gfCNCPoint5[16848] = {X 82.2240, Y 14.7584, Z -7.1667, A 0.000, B 0.000, C 0.000 }
gfCNCPoint5[16849] = {X 81.9226, Y 13.9083, Z -7.1667, A 0.000, B 0.000, C 0.000 }
gfCNCPoint5[16850] = {X 81.8152, Y 13.0128, Z -7.1667, A 0.000, B 0.000, C 0.000 }
gfCNCPoint5[16851] = {X 81.8151, Y 12.1868, Z -7.1667, A 0.000, B 0.000, C 0.000 }
gfCNCPoint5[16852] = {X 81.9174, Y 11.2789, Z -7.1667, A 0.000, B 0.000, C 0.000 }
gfCNCPoint5[16853] = {X 82.2191, Y 10.4166, Z -7.1667, A 0.000, B 0.000, C 0.000 }
gfCNCPoint5[16854] = {X 82.7052, Y 9.6430, Z -7.1667, A 0.000, B 0.000, C 0.000 }
gfCNCPoint5[16855] = {X 83.3512, Y 8.9969, Z -7.1667, A 0.000, B 0.000, C 0.000 }
gfCNCPoint5[16856] = {X 84.1248, Y 8.5109, Z -7.1667, A 0.000, B 0.000, C 0.000 }
gfCNCPoint5[16857] = {X 84.9872, Y 8.2091, Z -7.1667, A 0.000, B 0.000, C 0.000 }
gfCNCPoint5[16858] = {X 85.8951, Y 8.1068, Z -7.1667, A 0.000, B 0.000, C 0.000 }
gfCNCPoint5[16859] = {X 94.0497, Y 8.1068, Z -7.1667, A 0.000, B 0.000, C 0.000 }
gfCNCPoint5[16860] = {X 94.9576, Y 8.2091, Z -7.1667, A 0.000, B 0.000, C 0.000 }
gfCNCPoint5[16861] = {X 95.8199, Y 8.5109, Z -7.1667, A 0.000, B 0.000, C 0.000 }
gfCNCPoint5[16862] = {X 96.5935, Y 8.9969, Z -7.1667, A 0.000, B 0.000, C 0.000 }
gfCNCPoint5[16863] = {X 97.2395, Y 9.6430, Z -7.1667, A 0.000, B 0.000, C 0.000 }
gfCNCPoint5[16864] = {X 97.7256, Y 10.4166, Z -7.1667, A 0.000, B 0.000, C 0.000 }
gfCNCPoint5[16865] = {X 98.0274, Y 11.2789, Z -7.1667, A 0.000, B 0.000, C 0.000 }
gfCNCPoint5[16866] = {X 98.1297, Y 12.1868, Z -7.1667, A 0.000, B 0.000, C 0.000 }
gfCNCPoint5[16867] = {X 98.1297, Y 12.9782, Z -7.1667, A 0.000, B 0.000, C 0.000 }
gfCNCPoint5[16868] = {X 98.0632, Y 13.7116, Z -7.1667, A 0.000, B 0.000, C 0.000 }
gfCNCPoint5[16869] = {X 97.8659, Y 14.4211, Z -7.1667, A 0.000, B 0.000, C 0.000 }
gfCNCPoint5[16870] = {X 97.5443, Y 15.0836, Z -7.1667, A 0.000, B 0.000, C 0.000 }
gfCNCPoint5[16871] = {X 97.4977, Y 15.1591, Z -7.1667, A 0.000, B 0.000, C 0.000 }
gfCNCPoint5[16872] = {X 97.4495, Y 15.2336, Z -7.1667, A 0.000, B 0.000, C 0.000 }
gfCNCPoint5[16873] = {X 97.4864, Y 15.2810, Z -7.1667, A 0.000, B 0.000, C 0.000 }
gfCNCPoint5[16874] = {X 101.8776, Y 26.1666, Z -7.1667, A 0.000, B 0.000, C 0.000 }
gfCNCPoint5[16875] = {X 106.2844, Y 15.1969, Z -7.1667, A 0.000, B 0.000, C 0.000 }
gfCNCPoint5[16876] = {X 106.2408, Y 15.1282, Z -7.1667, A 0.000, B 0.000, C 0.000 }
gfCNCPoint5[16877] = {X 106.1986, Y 15.0586, Z -7.1667, A 0.000, B 0.000, C 0.000 }
gfCNCPoint5[16878] = {X 105.8896, Y 14.4146, Z -7.1667, A 0.000, B 0.000, C 0.000 }
gfCNCPoint5[16879] = {X 105.6975, Y 13.7266, Z -7.1667, A 0.000, B 0.000, C 0.000 }
gfCNCPoint5[16880] = {X 105.6285, Y 13.0157, Z -7.1667, A 0.000, B 0.000, C 0.000 }
gfCNCPoint5[16881] = {X 105.6283, Y 12.1868, Z -7.1667, A 0.000, B 0.000, C 0.000 }
gfCNCPoint5[16882] = {X 105.7306, Y 11.2789, Z -7.1667, A 0.000, B 0.000, C 0.000 }
gfCNCPoint5[16883] = {X 106.0323, Y 10.4166, Z -7.1667, A 0.000, B 0.000, C 0.000 }
gfCNCPoint5[16884] = {X 106.5184, Y 9.6430, Z -7.1667, A 0.000, B 0.000, C 0.000 }
gfCNCPoint5[16885] = {X 107.1644, Y 8.9969, Z -7.1667, A 0.000, B 0.000, C 0.000 }
gfCNCPoint5[16886] = {X 107.9380, Y 8.5109, Z -7.1667, A 0.000, B 0.000, C 0.000 }
gfCNCPoint5[16887] = {X 108.8004, Y 8.2091, Z -7.1667, A 0.000, B 0.000, C 0.000 }
gfCNCPoint5[16888] = {X 109.7083, Y 8.1068, Z -7.1667, A 0.000, B 0.000, C 0.000 }
gfCNCPoint5[16889] = {X 117.7916, Y 8.1068, Z -7.1667, A 0.000, B 0.000, C 0.000 }
gfCNCPoint5[16890] = {X 118.6995, Y 8.2091, Z -7.1667, A 0.000, B 0.000, C 0.000 }
gfCNCPoint5[16891] = {X 119.5618, Y 8.5109, Z -7.1667, A 0.000, B 0.000, C 0.000 }
gfCNCPoint5[16892] = {X 120.3354, Y 8.9969, Z -7.1667, A 0.000, B 0.000, C 0.000 }
gfCNCPoint5[16893] = {X 120.9814, Y 9.6430, Z -7.1667, A 0.000, B 0.000, C 0.000 }
gfCNCPoint5[16894] = {X 121.4675, Y 10.4166, Z -7.1667, A 0.000, B 0.000, C 0.000 }
gfCNCPoint5[16895] = {X 121.7693, Y 11.2789, Z -7.1667, A 0.000, B 0.000, C 0.000 }
gfCNCPoint5[16896] = {X 121.8716, Y 12.1868, Z -7.1667, A 0.000, B 0.000, C 0.000 }
gfCNCPoint5[16897] = {X 121.8716, Y 12.9782, Z -7.1667, A 0.000, B 0.000, C 0.000 }
gfCNCPoint5[16898] = {X 121.7699, Y 13.8830, Z -7.1667, A 0.000, B 0.000, C 0.000 }
gfCNCPoint5[16899] = {X 121.4702, Y 14.7427, Z -7.1667, A 0.000, B 0.000, C 0.000 }
gfCNCPoint5[16900] = {X 120.9872, Y 15.5146, Z -7.1667, A 0.000, B 0.000, C 0.000 }
gfCNCPoint5[16901] = {X 120.3451, Y 16.1601, Z -7.1667, A 0.000, B 0.000, C 0.000 }
gfCNCPoint5[16902] = {X 120.3450, Y 41.0278, Z -7.1667, A 0.000, B 0.000, C 0.000 }
gfCNCPoint5[16903] = {X 120.4677, Y 41.1291, Z -7.1667, A 0.000, B 0.000, C 0.000 }
gfCNCPoint5[16904] = {X 121.0553, Y 41.7605, Z -7.1667, A 0.000, B 0.000, C 0.000 }
gfCNCPoint5[16905] = {X 121.4971, Y 42.5013, Z -7.1667, A 0.000, B 0.000, C 0.000 }
gfCNCPoint5[16906] = {X 121.7732, Y 43.3184, Z -7.1667, A 0.000, B 0.000, C 0.000 }
gfCNCPoint5[16907] = {X 121.8714, Y 44.1754, Z -7.1667, A 0.000, B 0.000, C 0.000 }
gfCNCPoint5[16908] = {X 121.8716, Y 45.0000, Z -7.1667, A 0.000, B 0.000, C 0.000 }
gfCNCPoint5[16909] = {X 121.7693, Y 45.9079, Z -7.1667, A 0.000, B 0.000, C 0.000 }
gfCNCPoint5[16910] = {X 121.4675, Y 46.7702, Z -7.1667, A 0.000, B 0.000, C 0.000 }
gfCNCPoint5[16911] = {X 120.9814, Y 47.5438, Z -7.1667, A 0.000, B 0.000, C 0.000 }
gfCNCPoint5[16912] = {X 120.3354, Y 48.1899, Z -7.1667, A 0.000, B 0.000, C 0.000 }
gfCNCPoint5[16913] = {X 119.5618, Y 48.6760, Z -7.1667, A 0.000, B 0.000, C 0.000 }
gfCNCPoint5[16914] = {X 118.6995, Y 48.9777, Z -7.1667, A 0.000, B 0.000, C 0.000 }
gfCNCPoint5[16915] = {X 117.7916, Y 49.0800, Z -7.1667, A 0.000, B 0.000, C 0.000 }
gfCNCPoint5[16916] = {X 111.9185, Y 49.0800, Z -7.1667, A 0.000, B 0.000, C 0.000 }
gfCNCPoint5[16917] = {X 111.0151, Y 48.9787, Z -7.1667, A 0.000, B 0.000, C 0.000 }
gfCNCPoint5[16918] = {X 110.1565, Y 48.6799, Z -7.1667, A 0.000, B 0.000, C 0.000 }
gfCNCPoint5[16919] = {X 109.3855, Y 48.1985, Z -7.1667, A 0.000, B 0.000, C 0.000 }
gfCNCPoint5[16920] = {X 108.7401, Y 47.5582, Z -7.1667, A 0.000, B 0.000, C 0.000 }
gfCNCPoint5[16921] = {X 108.2526, Y 46.7909, Z -7.1667, A 0.000, B 0.000, C 0.000 }
gfCNCPoint5[16922] = {X 107.9470, Y 45.9348, Z -7.1667, A 0.000, B 0.000, C 0.000 }
gfCNCPoint5[16923] = {X 107.8386, Y 45.0322, Z -7.1667, A 0.000, B 0.000, C 0.000 }
gfCNCPoint5[16924] = {X 107.8385, Y 44.1771, Z -7.1667, A 0.000, B 0.000, C 0.000 }
gfCNCPoint5[16925] = {X 107.8717, Y 43.6680, Z -7.1667, A 0.000, B 0.000, C 0.000 }
gfCNCPoint5[16926] = {X 107.9710, Y 43.1676, Z -7.1667, A 0.000, B 0.000, C 0.000 }
gfCNCPoint5[16927] = {X 108.1299, Y 42.6955, Z -7.1667, A 0.000, B 0.000, C 0.000 }
gfCNCPoint5[16928] = {X 108.3475, Y 42.2474, Z -7.1667, A 0.000, B 0.000, C 0.000 }
gfCNCPoint5[16929] = {X 108.8090, Y 41.5687, Z -7.1667, A 0.000, B 0.000, C 0.000 }
gfCNCPoint5[16930] = {X 109.3649, Y 40.9650, Z -7.1667, A 0.000, B 0.000, C 0.000 }
gfCNCPoint5[16931] = {X 109.3648, Y 39.0029, Z -7.1667, A 0.000, B 0.000, C 0.000 }
gfCNCPoint5[16932] = {X 108.9865, Y 39.0029, Z -7.1667, A 0.000, B 0.000, C 0.000 }
gfCNCPoint5[16933] = {X 105.8902, Y 46.5692, Z -7.1667, A 0.000, B 0.000, C 0.000 }
gfCNCPoint5[16934] = {X 105.5407, Y 47.2300, Z -7.1667, A 0.000, B 0.000, C 0.000 }
gfCNCPoint5[16935] = {X 105.0765, Y 47.8159, Z -7.1667, A 0.000, B 0.000, C 0.000 }
gfCNCPoint5[16936] = {X 104.5133, Y 48.3073, Z -7.1667, A 0.000, B 0.000, C 0.000 }
gfCNCPoint5[16937] = {X 103.8698, Y 48.6877, Z -7.1667, A 0.000, B 0.000, C 0.000 }
gfCNCPoint5[16938] = {X 102.9784, Y 48.9895, Z -7.1667, A 0.000, B 0.000, C 0.000 }
gfCNCPoint5[16939] = {X 102.0417, Y 49.0792, Z -7.1667, A 0.000, B 0.000, C 0.000 }
gfCNCPoint5[16940] = {X 101.1093, Y 48.9518, Z -7.1667, A 0.000, B 0.000, C 0.000 }
gfCNCPoint5[16941] = {X 100.2309, Y 48.6142, Z -7.1667, A 0.000, B 0.000, C 0.000 }
gfCNCPoint5[16942] = {X 99.4532, Y 48.0843, Z -7.1667, A 0.000, B 0.000, C 0.000 }
gfCNCPoint5[16943] = {X 98.8176, Y 47.3903, Z -7.1667, A 0.000, B 0.000, C 0.000 }
gfCNCPoint5[16944] = {X 98.3579, Y 46.5692, Z -7.1667, A 0.000, B 0.000, C 0.000 }
gfCNCPoint5[16945] = {X 94.8929, Y 38.0952, Z -7.1667, A 0.000, B 0.000, C 0.000 }
gfCNCPoint5[16946] = {X 94.8920, Y 38.2309, Z -7.1667, A 0.000, B 0.000, C 0.000 }
gfCNCPoint5[16947] = {X 94.8920, Y 41.0165, Z -7.1667, A 0.000, B 0.000, C 0.000 }
gfCNCPoint5[16948] = {X 95.4369, Y 41.5527, Z -7.1667, A 0.000, B 0.000, C 0.000 }
gfCNCPoint5[16949] = {X 95.8744, Y 42.1796, Z -7.1667, A 0.000, B 0.000, C 0.000 }
gfCNCPoint5[16950] = {X 96.1092, Y 42.6624, Z -7.1667, A 0.000, B 0.000, C 0.000 }
gfCNCPoint5[16951] = {X 96.2799, Y 43.1714, Z -7.1667, A 0.000, B 0.000, C 0.000 }
gfCNCPoint5[16952] = {X 96.3820, Y 43.6855, Z -7.1667, A 0.000, B 0.000, C 0.000 }
gfCNCPoint5[16953] = {X 96.4185, Y 44.2083, Z -7.1667, A 0.000, B 0.000, C 0.000 }
gfCNCPoint5[16954] = {X 96.4184, Y 45.0392, Z -7.1667, A 0.000, B 0.000, C 0.000 }
gfCNCPoint5[16955] = {X 96.3086, Y 45.9406, Z -7.1667, A 0.000, B 0.000, C 0.000 }
gfCNCPoint5[16956] = {X 96.0023, Y 46.7954, Z -7.1667, A 0.000, B 0.000, C 0.000 }
gfCNCPoint5[16957] = {X 95.5144, Y 47.5613, Z -7.1667, A 0.000, B 0.000, C 0.000 }
gfCNCPoint5[16958] = {X 94.8692, Y 48.2003, Z -7.1667, A 0.000, B 0.000, C 0.000 }
gfCNCPoint5[16959] = {X 94.0987, Y 48.6808, Z -7.1667, A 0.000, B 0.000, C 0.000 }
gfCNCPoint5[16960] = {X 93.2410, Y 48.9789, Z -7.1667, A 0.000, B 0.000, C 0.000 }
gfCNCPoint5[16961] = {X 92.3385, Y 49.0800, Z -7.1667, A 0.000, B 0.000, C 0.000 }
gfCNCPoint5[16962] = {X 85.8951, Y 49.0800, Z -7.1667, A 0.000, B 0.000, C 0.000 }
gfCNCPoint5[16963] = {X 84.9918, Y 48.9788, Z -7.1667, A 0.000, B 0.000, C 0.000 }
gfCNCPoint5[16964] = {X 84.1334, Y 48.6801, Z -7.1667, A 0.000, B 0.000, C 0.000 }
gfCNCPoint5[16965] = {X 83.3624, Y 48.1987, Z -7.1667, A 0.000, B 0.000, C 0.000 }
gfCNCPoint5[16966] = {X 82.7171, Y 47.5586, Z -7.1667, A 0.000, B 0.000, C 0.000 }
gfCNCPoint5[16967] = {X 82.2295, Y 46.7916, Z -7.1667, A 0.000, B 0.000, C 0.000 }
gfCNCPoint5[16968] = {X 81.9238, Y 45.9356, Z -7.1667, A 0.000, B 0.000, C 0.000 }
gfCNCPoint5[16969] = {X 81.8152, Y 45.0332, Z -7.1667, A 0.000, B 0.000, C 0.000 }
gfCNCPoint5[16970] = {X 81.8151, Y 44.2084, Z -7.1667, A 0.000, B 0.000, C 0.000 }
gfCNCPoint5[16971] = {X 81.9200, Y 43.3034, Z -7.1667, A 0.000, B 0.000, C 0.000 }
gfCNCPoint5[16972] = {X 82.2207, Y 42.4433, Z -7.1667, A 0.000, B 0.000, C 0.000 }
gfCNCPoint5[16973] = {X 82.7024, Y 41.6699, Z -7.1667, A 0.000, B 0.000, C 0.000 }
gfCNCPoint5[16974] = {X 83.3419, Y 41.0209, Z -7.1667, A 0.000, B 0.000, C 0.000 }
gfCNCPoint5[16975] = {X 83.3418, Y 28.5910, Z -7.1667, A 0.000, B 0.000, C 0.000 }
gfCNCPoint5[16976] = {X 79.3418, Y 28.5910, Z -7.1667, A 0.000, B 0.000, C 0.000 }
gfCNCPoint5[16977] = {X 83.4218, Y 28.5910, Z -7.1667, A 0.000, B 0.000, C 0.000 }
gfCNCPoint5[16978] = {X 83.4217, Y 16.1216, Z -7.1667, A 0.000, B 0.000, C 0.000 }
gfCNCPoint5[16979] = {X 82.7800, Y 15.4873, Z -7.1667, A 0.000, B 0.000, C 0.000 }
gfCNCPoint5[16980] = {X 82.2969, Y 14.7253, Z -7.1667, A 0.000, B 0.000, C 0.000 }
gfCNCPoint5[16981] = {X 81.9968, Y 13.8745, Z -7.1667, A 0.000, B 0.000, C 0.000 }
gfCNCPoint5[16982] = {X 81.8951, Y 12.9780, Z -7.1667, A 0.000, B 0.000, C 0.000 }
gfCNCPoint5[16983] = {X 81.8951, Y 12.1868, Z -7.1667, A 0.000, B 0.000, C 0.000 }
gfCNCPoint5[16984] = {X 81.9954, Y 11.2967, Z -7.1667, A 0.000, B 0.000, C 0.000 }
gfCNCPoint5[16985] = {X 82.2912, Y 10.4513, Z -7.1667, A 0.000, B 0.000, C 0.000 }
gfCNCPoint5[16986] = {X 82.7677, Y 9.6929, Z -7.1667, A 0.000, B 0.000, C 0.000 }
gfCNCPoint5[16987] = {X 83.4011, Y 9.0595, Z -7.1667, A 0.000, B 0.000, C 0.000 }
gfCNCPoint5[16988] = {X 84.1595, Y 8.5829, Z -7.1667, A 0.000, B 0.000, C 0.000 }
gfCNCPoint5[16989] = {X 85.0050, Y 8.2871, Z -7.1667, A 0.000, B 0.000, C 0.000 }
gfCNCPoint5[16990] = {X 85.8951, Y 8.1868, Z -7.1667, A 0.000, B 0.000, C 0.000 }
gfCNCPoint5[16991] = {X 94.0497, Y 8.1868, Z -7.1667, A 0.000, B 0.000, C 0.000 }
gfCNCPoint5[16992] = {X 94.9398, Y 8.2871, Z -7.1667, A 0.000, B 0.000, C 0.000 }
gfCNCPoint5[16993] = {X 95.7852, Y 8.5829, Z -7.1667, A 0.000, B 0.000, C 0.000 }
gfCNCPoint5[16994] = {X 96.5436, Y 9.0595, Z -7.1667, A 0.000, B 0.000, C 0.000 }
gfCNCPoint5[16995] = {X 97.1770, Y 9.6929, Z -7.1667, A 0.000, B 0.000, C 0.000 }
gfCNCPoint5[16996] = {X 97.6535, Y 10.4513, Z -7.1667, A 0.000, B 0.000, C 0.000 }
gfCNCPoint5[16997] = {X 97.9494, Y 11.2967, Z -7.1667, A 0.000, B 0.000, C 0.000 }
gfCNCPoint5[16998] = {X 98.0497, Y 12.1868, Z -7.1667, A 0.000, B 0.000, C 0.000 }
gfCNCPoint5[16999] = {X 98.0495, Y 13.0192, Z -7.1667, A 0.000, B 0.000, C 0.000 }
gfCNCPoint5[17000] = {X 97.9795, Y 13.7241, Z -7.1667, A 0.000, B 0.000, C 0.000 }
gfCNCPoint5[17001] = {X 97.7862, Y 14.4056, Z -7.1667, A 0.000, B 0.000, C 0.000 }
gfCNCPoint5[17002] = {X 97.4758, Y 15.0424, Z -7.1667, A 0.000, B 0.000, C 0.000 }
gfCNCPoint5[17003] = {X 97.4132, Y 15.1429, Z -7.1667, A 0.000, B 0.000, C 0.000 }
gfCNCPoint5[17004] = {X 97.3476, Y 15.2415, Z -7.1667, A 0.000, B 0.000, C 0.000 }
gfCNCPoint5[17005] = {X 97.4122, Y 15.3109, Z -7.1667, A 0.000, B 0.000, C 0.000 }
gfCNCPoint5[17006] = {X 101.8768, Y 26.3785, Z -7.1667, A 0.000, B 0.000, C 0.000 }
gfCNCPoint5[17007] = {X 101.9496, Y 26.2020, Z -7.1667, A 0.000, B 0.000, C 0.000 }
gfCNCPoint5[17008] = {X 105.4120, Y 17.5683, Z -7.1667, A 0.000, B 0.000, C 0.000 }
gfCNCPoint5[17009] = {X 106.3409, Y 15.2554, Z -7.1667, A 0.000, B 0.000, C 0.000 }
gfCNCPoint5[17010] = {X 106.3813, Y 15.1986, Z -7.1667, A 0.000, B 0.000, C 0.000 }
gfCNCPoint5[17011] = {X 106.3231, Y 15.1090, Z -7.1667, A 0.000, B 0.000, C 0.000 }
gfCNCPoint5[17012] = {X 106.2675, Y 15.0178, Z -7.1667, A 0.000, B 0.000, C 0.000 }
gfCNCPoint5[17013] = {X 105.9601, Y 14.3749, Z -7.1667, A 0.000, B 0.000, C 0.000 }
gfCNCPoint5[17014] = {X 105.7717, Y 13.6877, Z -7.1667, A 0.000, B 0.000, C 0.000 }
gfCNCPoint5[17015] = {X 105.7083, Y 12.9780, Z -7.1667, A 0.000, B 0.000, C 0.000 }
gfCNCPoint5[17016] = {X 105.7083, Y 12.1868, Z -7.1667, A 0.000, B 0.000, C 0.000 }
gfCNCPoint5[17017] = {X 105.8086, Y 11.2967, Z -7.1667, A 0.000, B 0.000, C 0.000 }
gfCNCPoint5[17018] = {X 106.1044, Y 10.4513, Z -7.1667, A 0.000, B 0.000, C 0.000 }
gfCNCPoint5[17019] = {X 106.5810, Y 9.6929, Z -7.1667, A 0.000, B 0.000, C 0.000 }
gfCNCPoint5[17020] = {X 107.2143, Y 9.0595, Z -7.1667, A 0.000, B 0.000, C 0.000 }
gfCNCPoint5[17021] = {X 107.9727, Y 8.5829, Z -7.1667, A 0.000, B 0.000, C 0.000 }
gfCNCPoint5[17022] = {X 108.8182, Y 8.2871, Z -7.1667, A 0.000, B 0.000, C 0.000 }
gfCNCPoint5[17023] = {X 109.7083, Y 8.1868, Z -7.1667, A 0.000, B 0.000, C 0.000 }
gfCNCPoint5[17024] = {X 117.7916, Y 8.1868, Z -7.1667, A 0.000, B 0.000, C 0.000 }
gfCNCPoint5[17025] = {X 118.6817, Y 8.2871, Z -7.1667, A 0.000, B 0.000, C 0.000 }
gfCNCPoint5[17026] = {X 119.5271, Y 8.5829, Z -7.1667, A 0.000, B 0.000, C 0.000 }
gfCNCPoint5[17027] = {X 120.2855, Y 9.0595, Z -7.1667, A 0.000, B 0.000, C 0.000 }
gfCNCPoint5[17028] = {X 120.9189, Y 9.6929, Z -7.1667, A 0.000, B 0.000, C 0.000 }
gfCNCPoint5[17029] = {X 121.3955, Y 10.4513, Z -7.1667, A 0.000, B 0.000, C 0.000 }
gfCNCPoint5[17030] = {X 121.6913, Y 11.2967, Z -7.1667, A 0.000, B 0.000, C 0.000 }
gfCNCPoint5[17031] = {X 121.7916, Y 12.1868, Z -7.1667, A 0.000, B 0.000, C 0.000 }
gfCNCPoint5[17032] = {X 121.7914, Y 13.0192, Z -7.1667, A 0.000, B 0.000, C 0.000 }
gfCNCPoint5[17033] = {X 121.6828, Y 13.9045, Z -7.1667, A 0.000, B 0.000, C 0.000 }
gfCNCPoint5[17034] = {X 121.3807, Y 14.7438, Z -7.1667, A 0.000, B 0.000, C 0.000 }
gfCNCPoint5[17035] = {X 120.9002, Y 15.4952, Z -7.1667, A 0.000, B 0.000, C 0.000 }
gfCNCPoint5[17036] = {X 120.2651, Y 16.1215, Z -7.1667, A 0.000, B 0.000, C 0.000 }
gfCNCPoint5[17037] = {X 120.2650, Y 41.0655, Z -7.1667, A 0.000, B 0.000, C 0.000 }
gfCNCPoint5[17038] = {X 120.4160, Y 41.1901, Z -7.1667, A 0.000, B 0.000, C 0.000 }
gfCNCPoint5[17039] = {X 120.9967, Y 41.8157, Z -7.1667, A 0.000, B 0.000, C 0.000 }
gfCNCPoint5[17040] = {X 121.4315, Y 42.5502, Z -7.1667, A 0.000, B 0.000, C 0.000 }
gfCNCPoint5[17041] = {X 121.7005, Y 43.3602, Z -7.1667, A 0.000, B 0.000, C 0.000 }
gfCNCPoint5[17042] = {X 121.7916, Y 44.2089, Z -7.1667, A 0.000, B 0.000, C 0.000 }
gfCNCPoint5[17043] = {X 121.7916, Y 45.0000, Z -7.1667, A 0.000, B 0.000, C 0.000 }
gfCNCPoint5[17044] = {X 121.6913, Y 45.8901, Z -7.1667, A 0.000, B 0.000, C 0.000 }
gfCNCPoint5[17045] = {X 121.3955, Y 46.7355, Z -7.1667, A 0.000, B 0.000, C 0.000 }
gfCNCPoint5[17046] = {X 120.9189, Y 47.4940, Z -7.1667, A 0.000, B 0.000, C 0.000 }
gfCNCPoint5[17047] = {X 120.2855, Y 48.1273, Z -7.1667, A 0.000, B 0.000, C 0.000 }
gfCNCPoint5[17048] = {X 119.5271, Y 48.6039, Z -7.1667, A 0.000, B 0.000, C 0.000 }
gfCNCPoint5[17049] = {X 118.6817, Y 48.8997, Z -7.1667, A 0.000, B 0.000, C 0.000 }
gfCNCPoint5[17050] = {X 117.7916, Y 49.0000, Z -7.1667, A 0.000, B 0.000, C 0.000 }
gfCNCPoint5[17051] = {X 111.9185, Y 49.0000, Z -7.1667, A 0.000, B 0.000, C 0.000 }
gfCNCPoint5[17052] = {X 111.0284, Y 48.8997, Z -7.1667, A 0.000, B 0.000, C 0.000 }
gfCNCPoint5[17053] = {X 110.1829, Y 48.6039, Z -7.1667, A 0.000, B 0.000, C 0.000 }
gfCNCPoint5[17054] = {X 109.4245, Y 48.1273, Z -7.1667, A 0.000, B 0.000, C 0.000 }
gfCNCPoint5[17055] = {X 108.7911, Y 47.4939, Z -7.1667, A 0.000, B 0.000, C 0.000 }
gfCNCPoint5[17056] = {X 108.3146, Y 46.7355, Z -7.1667, A 0.000, B 0.000, C 0.000 }
gfCNCPoint5[17057] = {X 108.0188, Y 45.8901, Z -7.1667, A 0.000, B 0.000, C 0.000 }
gfCNCPoint5[17058] = {X 107.9185, Y 45.0000, Z -7.1667, A 0.000, B 0.000, C 0.000 }
gfCNCPoint5[17059] = {X 107.9185, Y 44.1771, Z -7.1667, A 0.000, B 0.000, C 0.000 }
gfCNCPoint5[17060] = {X 107.9511, Y 43.6784, Z -7.1667, A 0.000, B 0.000, C 0.000 }
gfCNCPoint5[17061] = {X 108.0483, Y 43.1883, Z -7.1667, A 0.000, B 0.000, C 0.000 }
gfCNCPoint5[17062] = {X 108.2039, Y 42.7258, Z -7.1667, A 0.000, B 0.000, C 0.000 }
gfCNCPoint5[17063] = {X 108.4171, Y 42.2868, Z -7.1667, A 0.000, B 0.000, C 0.000 }
gfCNCPoint5[17064] = {X 108.4423, Y 42.2431, Z -7.1667, A 0.000, B 0.000, C 0.000 }
gfCNCPoint5[17065] = {X 108.4680, Y 42.1997, Z -7.1667, A 0.000, B 0.000, C 0.000 }
gfCNCPoint5[17066] = {X 108.9141, Y 41.5653, Z -7.1667, A 0.000, B 0.000, C 0.000 }
gfCNCPoint5[17067] = {X 109.4449, Y 40.9999, Z -7.1667, A 0.000, B 0.000, C 0.000 }
gfCNCPoint5[17068] = {X 109.4448, Y 38.9229, Z -7.1667, A 0.000, B 0.000, C 0.000 }
gfCNCPoint5[17069] = {X 108.9328, Y 38.9229, Z -7.1667, A 0.000, B 0.000, C 0.000 }
gfCNCPoint5[17070] = {X 105.8164, Y 46.5384, Z -7.1667, A 0.000, B 0.000, C 0.000 }
gfCNCPoint5[17071] = {X 105.3339, Y 47.3869, Z -7.1667, A 0.000, B 0.000, C 0.000 }
gfCNCPoint5[17072] = {X 104.6602, Y 48.0932, Z -7.1667, A 0.000, B 0.000, C 0.000 }
gfCNCPoint5[17073] = {X 103.8355, Y 48.6154, Z -7.1667, A 0.000, B 0.000, C 0.000 }
gfCNCPoint5[17074] = {X 102.9580, Y 48.9121, Z -7.1667, A 0.000, B 0.000, C 0.000 }
gfCNCPoint5[17075] = {X 102.0357, Y 48.9990, Z -7.1667, A 0.000, B 0.000, C 0.000 }
gfCNCPoint5[17076] = {X 101.1182, Y 48.8715, Z -7.1667, A 0.000, B 0.000, C 0.000 }
gfCNCPoint5[17077] = {X 100.2546, Y 48.5362, Z -7.1667, A 0.000, B 0.000, C 0.000 }
gfCNCPoint5[17078] = {X 99.4912, Y 48.0114, Z -7.1667, A 0.000, B 0.000, C 0.000 }
gfCNCPoint5[17079] = {X 98.8691, Y 47.3250, Z -7.1667, A 0.000, B 0.000, C 0.000 }
gfCNCPoint5[17080] = {X 98.4216, Y 46.5139, Z -7.1667, A 0.000, B 0.000, C 0.000 }
gfCNCPoint5[17081] = {X 94.8156, Y 37.6948, Z -7.1667, A 0.000, B 0.000, C 0.000 }
gfCNCPoint5[17082] = {X 94.8120, Y 38.2306, Z -7.1667, A 0.000, B 0.000, C 0.000 }
gfCNCPoint5[17083] = {X 94.8120, Y 41.0546, Z -7.1667, A 0.000, B 0.000, C 0.000 }
gfCNCPoint5[17084] = {X 95.3635, Y 41.5899, Z -7.1667, A 0.000, B 0.000, C 0.000 }
gfCNCPoint5[17085] = {X 95.8049, Y 42.2191, Z -7.1667, A 0.000, B 0.000, C 0.000 }
gfCNCPoint5[17086] = {X 96.0352, Y 42.6926, Z -7.1667, A 0.000, B 0.000, C 0.000 }
gfCNCPoint5[17087] = {X 96.2026, Y 43.1919, Z -7.1667, A 0.000, B 0.000, C 0.000 }
gfCNCPoint5[17088] = {X 96.3027, Y 43.6961, Z -7.1667, A 0.000, B 0.000, C 0.000 }
gfCNCPoint5[17089] = {X 96.3385, Y 44.2089, Z -7.1667, A 0.000, B 0.000, C 0.000 }
gfCNCPoint5[17090] = {X 96.3384, Y 45.0384, Z -7.1667, A 0.000, B 0.000, C 0.000 }
gfCNCPoint5[17091] = {X 96.2308, Y 45.9222, Z -7.1667, A 0.000, B 0.000, C 0.000 }
gfCNCPoint5[17092] = {X 95.9304, Y 46.7602, Z -7.1667, A 0.000, B 0.000, C 0.000 }
gfCNCPoint5[17093] = {X 95.4521, Y 47.5111, Z -7.1667, A 0.000, B 0.000, C 0.000 }
gfCNCPoint5[17094] = {X 94.8196, Y 48.1376, Z -7.1667, A 0.000, B 0.000, C 0.000 }
gfCNCPoint5[17095] = {X 94.0642, Y 48.6086, Z -7.1667, A 0.000, B 0.000, C 0.000 }
gfCNCPoint5[17096] = {X 93.2233, Y 48.9009, Z -7.1667, A 0.000, B 0.000, C 0.000 }
gfCNCPoint5[17097] = {X 92.3385, Y 49.0000, Z -7.1667, A 0.000, B 0.000, C 0.000 }
gfCNCPoint5[17098] = {X 85.8951, Y 49.0000, Z -7.1667, A 0.000, B 0.000, C 0.000 }
gfCNCPoint5[17099] = {X 85.0050, Y 48.8997, Z -7.1667, A 0.000, B 0.000, C 0.000 }
gfCNCPoint5[17100] = {X 84.1595, Y 48.6039, Z -7.1667, A 0.000, B 0.000, C 0.000 }
gfCNCPoint5[17101] = {X 83.4011, Y 48.1273, Z -7.1667, A 0.000, B 0.000, C 0.000 }
gfCNCPoint5[17102] = {X 82.7677, Y 47.4939, Z -7.1667, A 0.000, B 0.000, C 0.000 }
gfCNCPoint5[17103] = {X 82.2912, Y 46.7355, Z -7.1667, A 0.000, B 0.000, C 0.000 }
gfCNCPoint5[17104] = {X 81.9954, Y 45.8901, Z -7.1667, A 0.000, B 0.000, C 0.000 }
gfCNCPoint5[17105] = {X 81.8951, Y 45.0000, Z -7.1667, A 0.000, B 0.000, C 0.000 }
gfCNCPoint5[17106] = {X 81.8951, Y 44.2088, Z -7.1667, A 0.000, B 0.000, C 0.000 }
gfCNCPoint5[17107] = {X 82.0001, Y 43.3120, Z -7.1667, A 0.000, B 0.000, C 0.000 }
gfCNCPoint5[17108] = {X 82.3011, Y 42.4607, Z -7.1667, A 0.000, B 0.000, C 0.000 }
gfCNCPoint5[17109] = {X 82.7829, Y 41.6972, Z -7.1667, A 0.000, B 0.000, C 0.000 }
gfCNCPoint5[17110] = {X 83.4219, Y 41.0592, Z -7.1667, A 0.000, B 0.000, C 0.000 }
gfCNCPoint5[17111] = {X 83.4218, Y 28.5910, Z -7.1667, A 0.000, B 0.000, C 0.000 }
gfCNCPoint5[17112] = {X 79.3418, Y 28.5910, Z -7.1667, A 0.000, B 0.000, C 0.000 }
gfCNCPoint5[17113] = {X 79.3418, Y 28.5910, Z -4.1667, A 0.000, B 0.000, C 0.000 }
gfCNCPoint5[17114] = {X 79.3418, Y 28.5910, Z 11.0000, A 0.000, B 0.000, C 0.000 }
gfCNCPoint5[17115] = {X 136.1636, Y 30.3969, Z 11.0000, A 0.000, B 0.000, C 0.000 }
gfCNCPoint5[17116] = {X 136.1636, Y 30.3969, Z -4.1667, A 0.000, B 0.000, C 0.000 }
gfCNCPoint5[17117] = {X 136.1636, Y 30.3969, Z -7.1667, A 0.000, B 0.000, C 0.000 }
gfCNCPoint5[17118] = {X 140.2436, Y 30.3969, Z -7.1667, A 0.000, B 0.000, C 0.000 }
gfCNCPoint5[17119] = {X 140.2436, Y 19.8782, Z -7.1667, A 0.000, B 0.000, C 0.000 }
gfCNCPoint5[17120] = {X 137.4233, Y 19.8779, Z -7.1667, A 0.000, B 0.000, C 0.000 }
gfCNCPoint5[17121] = {X 136.8909, Y 20.5223, Z -7.1667, A 0.000, B 0.000, C 0.000 }
gfCNCPoint5[17122] = {X 136.2444, Y 21.0521, Z -7.1667, A 0.000, B 0.000, C 0.000 }
gfCNCPoint5[17123] = {X 135.5079, Y 21.4475, Z -7.1667, A 0.000, B 0.000, C 0.000 }
gfCNCPoint5[17124] = {X 134.7091, Y 21.6937, Z -7.1667, A 0.000, B 0.000, C 0.000 }
gfCNCPoint5[17125] = {X 133.8778, Y 21.7814, Z -7.1667, A 0.000, B 0.000, C 0.000 }
gfCNCPoint5[17126] = {X 133.2006, Y 21.7815, Z -7.1667, A 0.000, B 0.000, C 0.000 }
gfCNCPoint5[17127] = {X 132.2394, Y 21.6732, Z -7.1667, A 0.000, B 0.000, C 0.000 }
gfCNCPoint5[17128] = {X 131.3263, Y 21.3537, Z -7.1667, A 0.000, B 0.000, C 0.000 }
gfCNCPoint5[17129] = {X 130.5072, Y 20.8390, Z -7.1667, A 0.000, B 0.000, C 0.000 }
gfCNCPoint5[17130] = {X 129.8231, Y 20.1550, Z -7.1667, A 0.000, B 0.000, C 0.000 }
gfCNCPoint5[17131] = {X 129.3085, Y 19.3359, Z -7.1667, A 0.000, B 0.000, C 0.000 }
gfCNCPoint5[17132] = {X 128.9890, Y 18.4228, Z -7.1667, A 0.000, B 0.000, C 0.000 }
gfCNCPoint5[17133] = {X 128.8806, Y 17.4615, Z -7.1667, A 0.000, B 0.000, C 0.000 }
gfCNCPoint5[17134] = {X 128.8806, Y 10.4835, Z -7.1667, A 0.000, B 0.000, C 0.000 }
gfCNCPoint5[17135] = {X 128.9874, Y 9.5289, Z -7.1667, A 0.000, B 0.000, C 0.000 }
gfCNCPoint5[17136] = {X 129.3026, Y 8.6214, Z -7.1667, A 0.000, B 0.000, C 0.000 }
gfCNCPoint5[17137] = {X 129.8104, Y 7.8061, Z -7.1667, A 0.000, B 0.000, C 0.000 }
gfCNCPoint5[17138] = {X 130.4859, Y 7.1231, Z -7.1667, A 0.000, B 0.000, C 0.000 }
gfCNCPoint5[17139] = {X 131.2956, Y 6.6063, Z -7.1667, A 0.000, B 0.000, C 0.000 }
gfCNCPoint5[17140] = {X 132.1995, Y 6.2811, Z -7.1667, A 0.000, B 0.000, C 0.000 }
gfCNCPoint5[17141] = {X 133.1529, Y 6.1638, Z -7.1667, A 0.000, B 0.000, C 0.000 }
gfCNCPoint5[17142] = {X 133.8866, Y 6.1637, Z -7.1667, A 0.000, B 0.000, C 0.000 }
gfCNCPoint5[17143] = {X 134.7108, Y 6.2517, Z -7.1667, A 0.000, B 0.000, C 0.000 }
gfCNCPoint5[17144] = {X 135.5031, Y 6.4955, Z -7.1667, A 0.000, B 0.000, C 0.000 }
gfCNCPoint5[17145] = {X 136.2342, Y 6.8861, Z -7.1667, A 0.000, B 0.000, C 0.000 }
gfCNCPoint5[17146] = {X 136.8772, Y 7.4091, Z -7.1667, A 0.000, B 0.000, C 0.000 }
gfCNCPoint5[17147] = {X 137.4085, Y 8.0454, Z -7.1667, A 0.000, B 0.000, C 0.000 }
gfCNCPoint5[17148] = {X 155.1133, Y 8.0467, Z -7.1667, A 0.000, B 0.000, C 0.000 }
gfCNCPoint5[17149] = {X 155.6453, Y 7.4093, Z -7.1667, A 0.000, B 0.000, C 0.000 }
gfCNCPoint5[17150] = {X 156.2894, Y 6.8855, Z -7.1667, A 0.000, B 0.000, C 0.000 }
gfCNCPoint5[17151] = {X 157.0219, Y 6.4946, Z -7.1667, A 0.000, B 0.000, C 0.000 }
gfCNCPoint5[17152] = {X 157.8156, Y 6.2510, Z -7.1667, A 0.000, B 0.000, C 0.000 }
gfCNCPoint5[17153] = {X 158.6412, Y 6.1637, Z -7.1667, A 0.000, B 0.000, C 0.000 }
gfCNCPoint5[17154] = {X 159.3781, Y 6.1639, Z -7.1667, A 0.000, B 0.000, C 0.000 }
gfCNCPoint5[17155] = {X 160.3301, Y 6.2828, Z -7.1667, A 0.000, B 0.000, C 0.000 }
gfCNCPoint5[17156] = {X 161.2324, Y 6.6088, Z -7.1667, A 0.000, B 0.000, C 0.000 }
gfCNCPoint5[17157] = {X 162.0405, Y 7.1260, Z -7.1667, A 0.000, B 0.000, C 0.000 }
gfCNCPoint5[17158] = {X 162.7145, Y 7.8088, Z -7.1667, A 0.000, B 0.000, C 0.000 }
gfCNCPoint5[17159] = {X 163.2212, Y 8.6236, Z -7.1667, A 0.000, B 0.000, C 0.000 }
gfCNCPoint5[17160] = {X 163.5355, Y 9.5300, Z -7.1667, A 0.000, B 0.000, C 0.000 }
gfCNCPoint5[17161] = {X 163.6421, Y 10.4835, Z -7.1667, A 0.000, B 0.000, C 0.000 }
gfCNCPoint5[17162] = {X 163.6421, Y 17.4615, Z -7.1667, A 0.000, B 0.000, C 0.000 }
gfCNCPoint5[17163] = {X 163.5355, Y 18.4152, Z -7.1667, A 0.000, B 0.000, C 0.000 }
gfCNCPoint5[17164] = {X 163.2211, Y 19.3218, Z -7.1667, A 0.000, B 0.000, C 0.000 }
gfCNCPoint5[17165] = {X 162.7142, Y 20.1366, Z -7.1667, A 0.000, B 0.000, C 0.000 }
gfCNCPoint5[17166] = {X 162.0400, Y 20.8194, Z -7.1667, A 0.000, B 0.000, C 0.000 }
gfCNCPoint5[17167] = {X 161.2318, Y 21.3365, Z -7.1667, A 0.000, B 0.000, C 0.000 }
gfCNCPoint5[17168] = {X 160.3292, Y 21.6625, Z -7.1667, A 0.000, B 0.000, C 0.000 }
gfCNCPoint5[17169] = {X 159.3770, Y 21.7812, Z -7.1667, A 0.000, B 0.000, C 0.000 }
gfCNCPoint5[17170] = {X 158.6794, Y 21.7815, Z -7.1667, A 0.000, B 0.000, C 0.000 }
gfCNCPoint5[17171] = {X 157.8410, Y 21.6970, Z -7.1667, A 0.000, B 0.000, C 0.000 }
gfCNCPoint5[17172] = {X 157.0346, Y 21.4525, Z -7.1667, A 0.000, B 0.000, C 0.000 }
gfCNCPoint5[17173] = {X 156.2904, Y 21.0570, Z -7.1667, A 0.000, B 0.000, C 0.000 }
gfCNCPoint5[17174] = {X 155.6365, Y 20.5255, Z -7.1667, A 0.000, B 0.000, C 0.000 }
gfCNCPoint5[17175] = {X 155.0973, Y 19.8779, Z -7.1667, A 0.000, B 0.000, C 0.000 }
gfCNCPoint5[17176] = {X 152.2772, Y 19.8789, Z -7.1667, A 0.000, B 0.000, C 0.000 }
gfCNCPoint5[17177] = {X 152.2761, Y 40.8742, Z -7.1667, A 0.000, B 0.000, C 0.000 }
gfCNCPoint5[17178] = {X 152.7408, Y 41.3745, Z -7.1667, A 0.000, B 0.000, C 0.000 }
gfCNCPoint5[17179] = {X 152.8367, Y 41.4887, Z -7.1667, A 0.000, B 0.000, C 0.000 }
gfCNCPoint5[17180] = {X 153.3624, Y 42.3140, Z -7.1667, A 0.000, B 0.000, C 0.000 }
gfCNCPoint5[17181] = {X 153.6900, Y 43.2360, Z -7.1667, A 0.000, B 0.000, C 0.000 }
gfCNCPoint5[17182] = {X 153.8031, Y 44.2079, Z -7.1667, A 0.000, B 0.000, C 0.000 }
gfCNCPoint5[17183] = {X 153.8029, Y 45.0415, Z -7.1667, A 0.000, B 0.000, C 0.000 }
gfCNCPoint5[17184] = {X 153.6867, Y 45.9960, Z -7.1667, A 0.000, B 0.000, C 0.000 }
gfCNCPoint5[17185] = {X 153.3623, Y 46.9011, Z -7.1667, A 0.000, B 0.000, C 0.000 }
gfCNCPoint5[17186] = {X 152.8458, Y 47.7120, Z -7.1667, A 0.000, B 0.000, C 0.000 }
gfCNCPoint5[17187] = {X 152.1626, Y 48.3886, Z -7.1667, A 0.000, B 0.000, C 0.000 }
gfCNCPoint5[17188] = {X 151.3468, Y 48.8973, Z -7.1667, A 0.000, B 0.000, C 0.000 }
gfCNCPoint5[17189] = {X 150.4386, Y 49.2130, Z -7.1667, A 0.000, B 0.000, C 0.000 }
gfCNCPoint5[17190] = {X 149.4831, Y 49.3200, Z -7.1667, A 0.000, B 0.000, C 0.000 }
gfCNCPoint5[17191] = {X 143.0396, Y 49.3200, Z -7.1667, A 0.000, B 0.000, C 0.000 }
gfCNCPoint5[17192] = {X 142.0831, Y 49.2128, Z -7.1667, A 0.000, B 0.000, C 0.000 }
gfCNCPoint5[17193] = {X 141.1741, Y 48.8964, Z -7.1667, A 0.000, B 0.000, C 0.000 }
gfCNCPoint5[17194] = {X 140.3576, Y 48.3866, Z -7.1667, A 0.000, B 0.000, C 0.000 }
gfCNCPoint5[17195] = {X 139.6743, Y 47.7087, Z -7.1667, A 0.000, B 0.000, C 0.000 }
gfCNCPoint5[17196] = {X 139.1581, Y 46.8964, Z -7.1667, A 0.000, B 0.000, C 0.000 }
gfCNCPoint5[17197] = {X 138.8346, Y 45.9899, Z -7.1667, A 0.000, B 0.000, C 0.000 }
gfCNCPoint5[17198] = {X 138.7198, Y 45.0342, Z -7.1667, A 0.000, B 0.000, C 0.000 }
gfCNCPoint5[17199] = {X 138.7200, Y 44.1494, Z -7.1667, A 0.000, B 0.000, C 0.000 }
gfCNCPoint5[17200] = {X 138.8305, Y 43.2364, Z -7.1667, A 0.000, B 0.000, C 0.000 }
gfCNCPoint5[17201] = {X 139.1317, Y 42.3675, Z -7.1667, A 0.000, B 0.000, C 0.000 }
gfCNCPoint5[17202] = {X 139.6099, Y 41.5821, Z -7.1667, A 0.000, B 0.000, C 0.000 }
gfCNCPoint5[17203] = {X 140.2436, Y 40.9157, Z -7.1667, A 0.000, B 0.000, C 0.000 }
gfCNCPoint5[17204] = {X 140.2436, Y 30.3969, Z -7.1667, A 0.000, B 0.000, C 0.000 }
gfCNCPoint5[17205] = {X 136.2436, Y 30.3969, Z -7.1667, A 0.000, B 0.000, C 0.000 }
gfCNCPoint5[17206] = {X 140.3236, Y 30.3969, Z -7.1667, A 0.000, B 0.000, C 0.000 }
gfCNCPoint5[17207] = {X 140.3236, Y 19.7982, Z -7.1667, A 0.000, B 0.000, C 0.000 }
gfCNCPoint5[17208] = {X 137.3793, Y 19.7979, Z -7.1667, A 0.000, B 0.000, C 0.000 }
gfCNCPoint5[17209] = {X 137.3564, Y 19.8340, Z -7.1667, A 0.000, B 0.000, C 0.000 }
gfCNCPoint5[17210] = {X 136.8339, Y 20.4662, Z -7.1667, A 0.000, B 0.000, C 0.000 }
gfCNCPoint5[17211] = {X 136.1994, Y 20.9860, Z -7.1667, A 0.000, B 0.000, C 0.000 }
gfCNCPoint5[17212] = {X 135.4767, Y 21.3739, Z -7.1667, A 0.000, B 0.000, C 0.000 }
gfCNCPoint5[17213] = {X 134.6928, Y 21.6154, Z -7.1667, A 0.000, B 0.000, C 0.000 }
gfCNCPoint5[17214] = {X 133.8772, Y 21.7014, Z -7.1667, A 0.000, B 0.000, C 0.000 }
gfCNCPoint5[17215] = {X 133.2006, Y 21.7015, Z -7.1667, A 0.000, B 0.000, C 0.000 }
gfCNCPoint5[17216] = {X 132.2572, Y 21.5952, Z -7.1667, A 0.000, B 0.000, C 0.000 }
gfCNCPoint5[17217] = {X 131.3610, Y 21.2816, Z -7.1667, A 0.000, B 0.000, C 0.000 }
gfCNCPoint5[17218] = {X 130.5570, Y 20.7765, Z -7.1667, A 0.000, B 0.000, C 0.000 }
gfCNCPoint5[17219] = {X 129.8857, Y 20.1051, Z -7.1667, A 0.000, B 0.000, C 0.000 }
gfCNCPoint5[17220] = {X 129.3805, Y 19.3012, Z -7.1667, A 0.000, B 0.000, C 0.000 }
gfCNCPoint5[17221] = {X 129.0669, Y 18.4050, Z -7.1667, A 0.000, B 0.000, C 0.000 }
gfCNCPoint5[17222] = {X 128.9606, Y 17.4615, Z -7.1667, A 0.000, B 0.000, C 0.000 }
gfCNCPoint5[17223] = {X 128.9606, Y 10.4835, Z -7.1667, A 0.000, B 0.000, C 0.000 }
gfCNCPoint5[17224] = {X 129.0655, Y 9.5466, Z -7.1667, A 0.000, B 0.000, C 0.000 }
gfCNCPoint5[17225] = {X 129.3747, Y 8.6559, Z -7.1667, A 0.000, B 0.000, C 0.000 }
gfCNCPoint5[17226] = {X 129.8732, Y 7.8557, Z -7.1667, A 0.000, B 0.000, C 0.000 }
gfCNCPoint5[17227] = {X 130.5362, Y 7.1853, Z -7.1667, A 0.000, B 0.000, C 0.000 }
gfCNCPoint5[17228] = {X 131.3309, Y 6.6781, Z -7.1667, A 0.000, B 0.000, C 0.000 }
gfCNCPoint5[17229] = {X 132.2180, Y 6.3589, Z -7.1667, A 0.000, B 0.000, C 0.000 }
gfCNCPoint5[17230] = {X 133.1538, Y 6.2438, Z -7.1667, A 0.000, B 0.000, C 0.000 }
gfCNCPoint5[17231] = {X 133.8858, Y 6.2437, Z -7.1667, A 0.000, B 0.000, C 0.000 }
gfCNCPoint5[17232] = {X 134.7030, Y 6.3318, Z -7.1667, A 0.000, B 0.000, C 0.000 }
gfCNCPoint5[17233] = {X 135.4878, Y 6.5758, Z -7.1667, A 0.000, B 0.000, C 0.000 }
gfCNCPoint5[17234] = {X 136.2108, Y 6.9668, Z -7.1667, A 0.000, B 0.000, C 0.000 }
gfCNCPoint5[17235] = {X 136.8449, Y 7.4898, Z -7.1667, A 0.000, B 0.000, C 0.000 }
gfCNCPoint5[17236] = {X 137.3660, Y 8.1254, Z -7.1667, A 0.000, B 0.000, C 0.000 }
gfCNCPoint5[17237] = {X 155.1558, Y 8.1267, Z -7.1667, A 0.000, B 0.000, C 0.000 }
gfCNCPoint5[17238] = {X 155.6777, Y 7.4900, Z -7.1667, A 0.000, B 0.000, C 0.000 }
gfCNCPoint5[17239] = {X 156.3127, Y 6.9662, Z -7.1667, A 0.000, B 0.000, C 0.000 }
gfCNCPoint5[17240] = {X 157.0371, Y 6.5749, Z -7.1667, A 0.000, B 0.000, C 0.000 }
gfCNCPoint5[17241] = {X 157.8234, Y 6.3310, Z -7.1667, A 0.000, B 0.000, C 0.000 }
gfCNCPoint5[17242] = {X 158.6420, Y 6.2437, Z -7.1667, A 0.000, B 0.000, C 0.000 }
gfCNCPoint5[17243] = {X 159.3770, Y 6.2439, Z -7.1667, A 0.000, B 0.000, C 0.000 }
gfCNCPoint5[17244] = {X 160.3114, Y 6.3606, Z -7.1667, A 0.000, B 0.000, C 0.000 }
gfCNCPoint5[17245] = {X 161.1970, Y 6.6806, Z -7.1667, A 0.000, B 0.000, C 0.000 }
gfCNCPoint5[17246] = {X 161.9902, Y 7.1882, Z -7.1667, A 0.000, B 0.000, C 0.000 }
gfCNCPoint5[17247] = {X 162.6517, Y 7.8584, Z -7.1667, A 0.000, B 0.000, C 0.000 }
gfCNCPoint5[17248] = {X 163.1490, Y 8.6580, Z -7.1667, A 0.000, B 0.000, C 0.000 }
gfCNCPoint5[17249] = {X 163.4575, Y 9.5477, Z -7.1667, A 0.000, B 0.000, C 0.000 }
gfCNCPoint5[17250] = {X 163.5621, Y 10.4835, Z -7.1667, A 0.000, B 0.000, C 0.000 }
gfCNCPoint5[17251] = {X 163.5621, Y 17.4615, Z -7.1667, A 0.000, B 0.000, C 0.000 }
gfCNCPoint5[17252] = {X 163.4575, Y 18.3975, Z -7.1667, A 0.000, B 0.000, C 0.000 }
gfCNCPoint5[17253] = {X 163.1489, Y 19.2873, Z -7.1667, A 0.000, B 0.000, C 0.000 }
gfCNCPoint5[17254] = {X 162.6514, Y 20.0870, Z -7.1667, A 0.000, B 0.000, C 0.000 }
gfCNCPoint5[17255] = {X 161.9897, Y 20.7572, Z -7.1667, A 0.000, B 0.000, C 0.000 }
gfCNCPoint5[17256] = {X 161.1964, Y 21.2648, Z -7.1667, A 0.000, B 0.000, C 0.000 }
gfCNCPoint5[17257] = {X 160.3106, Y 21.5847, Z -7.1667, A 0.000, B 0.000, C 0.000 }
gfCNCPoint5[17258] = {X 159.3760, Y 21.7012, Z -7.1667, A 0.000, B 0.000, C 0.000 }
gfCNCPoint5[17259] = {X 158.6797, Y 21.7015, Z -7.1667, A 0.000, B 0.000, C 0.000 }
gfCNCPoint5[17260] = {X 157.8484, Y 21.6169, Z -7.1667, A 0.000, B 0.000, C 0.000 }
gfCNCPoint5[17261] = {X 157.0495, Y 21.3721, Z -7.1667, A 0.000, B 0.000, C 0.000 }
gfCNCPoint5[17262] = {X 156.3136, Y 20.9763, Z -7.1667, A 0.000, B 0.000, C 0.000 }
gfCNCPoint5[17263] = {X 155.6688, Y 20.4448, Z -7.1667, A 0.000, B 0.000, C 0.000 }
gfCNCPoint5[17264] = {X 155.1399, Y 19.7979, Z -7.1667, A 0.000, B 0.000, C 0.000 }
gfCNCPoint5[17265] = {X 152.1972, Y 19.7989, Z -7.1667, A 0.000, B 0.000, C 0.000 }
gfCNCPoint5[17266] = {X 152.1961, Y 40.9056, Z -7.1667, A 0.000, B 0.000, C 0.000 }
gfCNCPoint5[17267] = {X 152.6808, Y 41.4275, Z -7.1667, A 0.000, B 0.000, C 0.000 }
gfCNCPoint5[17268] = {X 152.7750, Y 41.5396, Z -7.1667, A 0.000, B 0.000, C 0.000 }
gfCNCPoint5[17269] = {X 153.2907, Y 42.3495, Z -7.1667, A 0.000, B 0.000, C 0.000 }
gfCNCPoint5[17270] = {X 153.6122, Y 43.2543, Z -7.1667, A 0.000, B 0.000, C 0.000 }
gfCNCPoint5[17271] = {X 153.7231, Y 44.2081, Z -7.1667, A 0.000, B 0.000, C 0.000 }
gfCNCPoint5[17272] = {X 153.7229, Y 45.0408, Z -7.1667, A 0.000, B 0.000, C 0.000 }
gfCNCPoint5[17273] = {X 153.6089, Y 45.9775, Z -7.1667, A 0.000, B 0.000, C 0.000 }
gfCNCPoint5[17274] = {X 153.2905, Y 46.8659, Z -7.1667, A 0.000, B 0.000, C 0.000 }
gfCNCPoint5[17275] = {X 152.7835, Y 47.6618, Z -7.1667, A 0.000, B 0.000, C 0.000 }
gfCNCPoint5[17276] = {X 152.1130, Y 48.3258, Z -7.1667, A 0.000, B 0.000, C 0.000 }
gfCNCPoint5[17277] = {X 151.3123, Y 48.8251, Z -7.1667, A 0.000, B 0.000, C 0.000 }
gfCNCPoint5[17278] = {X 150.4209, Y 49.1350, Z -7.1667, A 0.000, B 0.000, C 0.000 }
gfCNCPoint5[17279] = {X 149.4831, Y 49.2400, Z -7.1667, A 0.000, B 0.000, C 0.000 }
gfCNCPoint5[17280] = {X 143.0396, Y 49.2400, Z -7.1667, A 0.000, B 0.000, C 0.000 }
gfCNCPoint5[17281] = {X 142.1008, Y 49.1348, Z -7.1667, A 0.000, B 0.000, C 0.000 }
gfCNCPoint5[17282] = {X 141.2086, Y 48.8243, Z -7.1667, A 0.000, B 0.000, C 0.000 }
gfCNCPoint5[17283] = {X 140.4073, Y 48.3239, Z -7.1667, A 0.000, B 0.000, C 0.000 }
gfCNCPoint5[17284] = {X 139.7367, Y 47.6586, Z -7.1667, A 0.000, B 0.000, C 0.000 }
gfCNCPoint5[17285] = {X 139.2300, Y 46.8612, Z -7.1667, A 0.000, B 0.000, C 0.000 }
gfCNCPoint5[17286] = {X 138.9124, Y 45.9715, Z -7.1667, A 0.000, B 0.000, C 0.000 }
gfCNCPoint5[17287] = {X 138.7998, Y 45.0336, Z -7.1667, A 0.000, B 0.000, C 0.000 }
gfCNCPoint5[17288] = {X 138.8000, Y 44.1505, Z -7.1667, A 0.000, B 0.000, C 0.000 }
gfCNCPoint5[17289] = {X 138.9105, Y 43.2454, Z -7.1667, A 0.000, B 0.000, C 0.000 }
gfCNCPoint5[17290] = {X 139.2119, Y 42.3850, Z -7.1667, A 0.000, B 0.000, C 0.000 }
gfCNCPoint5[17291] = {X 139.6903, Y 41.6088, Z -7.1667, A 0.000, B 0.000, C 0.000 }
gfCNCPoint5[17292] = {X 140.3236, Y 40.9529, Z -7.1667, A 0.000, B 0.000, C 0.000 }
gfCNCPoint5[17293] = {X 140.3236, Y 30.3969, Z -7.1667, A 0.000, B 0.000, C 0.000 }
gfCNCPoint5[17294] = {X 136.3236, Y 30.3969, Z -7.1667, A 0.000, B 0.000, C 0.000 }
gfCNCPoint5[17295] = {X 140.4036, Y 30.3969, Z -7.1667, A 0.000, B 0.000, C 0.000 }
gfCNCPoint5[17296] = {X 140.4036, Y 19.7182, Z -7.1667, A 0.000, B 0.000, C 0.000 }
gfCNCPoint5[17297] = {X 137.3352, Y 19.7179, Z -7.1667, A 0.000, B 0.000, C 0.000 }
gfCNCPoint5[17298] = {X 137.2894, Y 19.7903, Z -7.1667, A 0.000, B 0.000, C 0.000 }
gfCNCPoint5[17299] = {X 136.7767, Y 20.4102, Z -7.1667, A 0.000, B 0.000, C 0.000 }
gfCNCPoint5[17300] = {X 136.1543, Y 20.9199, Z -7.1667, A 0.000, B 0.000, C 0.000 }
gfCNCPoint5[17301] = {X 135.4454, Y 21.3002, Z -7.1667, A 0.000, B 0.000, C 0.000 }
gfCNCPoint5[17302] = {X 134.6766, Y 21.5370, Z -7.1667, A 0.000, B 0.000, C 0.000 }
gfCNCPoint5[17303] = {X 133.8765, Y 21.6214, Z -7.1667, A 0.000, B 0.000, C 0.000 }
gfCNCPoint5[17304] = {X 133.2006, Y 21.6215, Z -7.1667, A 0.000, B 0.000, C 0.000 }
gfCNCPoint5[17305] = {X 132.2750, Y 21.5172, Z -7.1667, A 0.000, B 0.000, C 0.000 }
gfCNCPoint5[17306] = {X 131.3957, Y 21.2096, Z -7.1667, A 0.000, B 0.000, C 0.000 }
gfCNCPoint5[17307] = {X 130.6069, Y 20.7140, Z -7.1667, A 0.000, B 0.000, C 0.000 }
gfCNCPoint5[17308] = {X 129.9482, Y 20.0553, Z -7.1667, A 0.000, B 0.000, C 0.000 }
gfCNCPoint5[17309] = {X 129.4526, Y 19.2665, Z -7.1667, A 0.000, B 0.000, C 0.000 }
gfCNCPoint5[17310] = {X 129.1449, Y 18.3872, Z -7.1667, A 0.000, B 0.000, C 0.000 }
gfCNCPoint5[17311] = {X 129.0406, Y 17.4615, Z -7.1667, A 0.000, B 0.000, C 0.000 }
gfCNCPoint5[17312] = {X 129.0406, Y 10.4835, Z -7.1667, A 0.000, B 0.000, C 0.000 }
gfCNCPoint5[17313] = {X 129.1435, Y 9.5642, Z -7.1667, A 0.000, B 0.000, C 0.000 }
gfCNCPoint5[17314] = {X 129.4469, Y 8.6904, Z -7.1667, A 0.000, B 0.000, C 0.000 }
gfCNCPoint5[17315] = {X 129.9360, Y 7.9052, Z -7.1667, A 0.000, B 0.000, C 0.000 }
gfCNCPoint5[17316] = {X 130.5864, Y 7.2475, Z -7.1667, A 0.000, B 0.000, C 0.000 }
gfCNCPoint5[17317] = {X 131.3662, Y 6.7499, Z -7.1667, A 0.000, B 0.000, C 0.000 }
gfCNCPoint5[17318] = {X 132.2366, Y 6.4368, Z -7.1667, A 0.000, B 0.000, C 0.000 }
gfCNCPoint5[17319] = {X 133.1547, Y 6.3238, Z -7.1667, A 0.000, B 0.000, C 0.000 }
gfCNCPoint5[17320] = {X 133.8850, Y 6.3237, Z -7.1667, A 0.000, B 0.000, C 0.000 }
gfCNCPoint5[17321] = {X 134.6951, Y 6.4119, Z -7.1667, A 0.000, B 0.000, C 0.000 }
gfCNCPoint5[17322] = {X 135.4725, Y 6.6562, Z -7.1667, A 0.000, B 0.000, C 0.000 }
gfCNCPoint5[17323] = {X 136.1873, Y 7.0474, Z -7.1667, A 0.000, B 0.000, C 0.000 }
gfCNCPoint5[17324] = {X 136.8122, Y 7.5705, Z -7.1667, A 0.000, B 0.000, C 0.000 }
gfCNCPoint5[17325] = {X 137.3231, Y 8.2054, Z -7.1667, A 0.000, B 0.000, C 0.000 }
gfCNCPoint5[17326] = {X 155.1988, Y 8.2067, Z -7.1667, A 0.000, B 0.000, C 0.000 }
gfCNCPoint5[17327] = {X 155.7103, Y 7.5707, Z -7.1667, A 0.000, B 0.000, C 0.000 }
gfCNCPoint5[17328] = {X 156.3362, Y 7.0469, Z -7.1667, A 0.000, B 0.000, C 0.000 }
gfCNCPoint5[17329] = {X 157.0524, Y 6.6553, Z -7.1667, A 0.000, B 0.000, C 0.000 }
gfCNCPoint5[17330] = {X 157.8312, Y 6.4111, Z -7.1667, A 0.000, B 0.000, C 0.000 }
gfCNCPoint5[17331] = {X 158.6427, Y 6.3237, Z -7.1667, A 0.000, B 0.000, C 0.000 }
gfCNCPoint5[17332] = {X 159.3760, Y 6.3239, Z -7.1667, A 0.000, B 0.000, C 0.000 }
gfCNCPoint5[17333] = {X 160.2928, Y 6.4383, Z -7.1667, A 0.000, B 0.000, C 0.000 }
gfCNCPoint5[17334] = {X 161.1617, Y 6.7524, Z -7.1667, A 0.000, B 0.000, C 0.000 }
gfCNCPoint5[17335] = {X 161.9398, Y 7.2504, Z -7.1667, A 0.000, B 0.000, C 0.000 }
gfCNCPoint5[17336] = {X 162.5889, Y 7.9079, Z -7.1667, A 0.000, B 0.000, C 0.000 }
gfCNCPoint5[17337] = {X 163.0768, Y 8.6925, Z -7.1667, A 0.000, B 0.000, C 0.000 }
gfCNCPoint5[17338] = {X 163.3795, Y 9.5653, Z -7.1667, A 0.000, B 0.000, C 0.000 }
gfCNCPoint5[17339] = {X 163.4821, Y 10.4835, Z -7.1667, A 0.000, B 0.000, C 0.000 }
gfCNCPoint5[17340] = {X 163.4821, Y 17.4615, Z -7.1667, A 0.000, B 0.000, C 0.000 }
gfCNCPoint5[17341] = {X 163.3795, Y 18.3798, Z -7.1667, A 0.000, B 0.000, C 0.000 }
gfCNCPoint5[17342] = {X 163.0767, Y 19.2527, Z -7.1667, A 0.000, B 0.000, C 0.000 }
gfCNCPoint5[17343] = {X 162.5887, Y 20.0373, Z -7.1667, A 0.000, B 0.000, C 0.000 }
gfCNCPoint5[17344] = {X 161.9396, Y 20.6948, Z -7.1667, A 0.000, B 0.000, C 0.000 }
gfCNCPoint5[17345] = {X 161.1613, Y 21.1929, Z -7.1667, A 0.000, B 0.000, C 0.000 }
gfCNCPoint5[17346] = {X 160.2923, Y 21.5068, Z -7.1667, A 0.000, B 0.000, C 0.000 }
gfCNCPoint5[17347] = {X 159.3755, Y 21.6212, Z -7.1667, A 0.000, B 0.000, C 0.000 }
gfCNCPoint5[17348] = {X 158.6799, Y 21.6215, Z -7.1667, A 0.000, B 0.000, C 0.000 }
gfCNCPoint5[17349] = {X 157.8559, Y 21.5368, Z -7.1667, A 0.000, B 0.000, C 0.000 }
gfCNCPoint5[17350] = {X 157.0645, Y 21.2916, Z -7.1667, A 0.000, B 0.000, C 0.000 }
gfCNCPoint5[17351] = {X 156.3369, Y 20.8955, Z -7.1667, A 0.000, B 0.000, C 0.000 }
gfCNCPoint5[17352] = {X 155.7015, Y 20.3640, Z -7.1667, A 0.000, B 0.000, C 0.000 }
gfCNCPoint5[17353] = {X 155.1830, Y 19.7179, Z -7.1667, A 0.000, B 0.000, C 0.000 }
gfCNCPoint5[17354] = {X 152.1172, Y 19.7189, Z -7.1667, A 0.000, B 0.000, C 0.000 }
gfCNCPoint5[17355] = {X 152.1161, Y 40.9370, Z -7.1667, A 0.000, B 0.000, C 0.000 }
gfCNCPoint5[17356] = {X 152.6209, Y 41.4805, Z -7.1667, A 0.000, B 0.000, C 0.000 }
gfCNCPoint5[17357] = {X 152.7132, Y 41.5904, Z -7.1667, A 0.000, B 0.000, C 0.000 }
gfCNCPoint5[17358] = {X 153.2191, Y 42.3851, Z -7.1667, A 0.000, B 0.000, C 0.000 }
gfCNCPoint5[17359] = {X 153.5343, Y 43.2727, Z -7.1667, A 0.000, B 0.000, C 0.000 }
gfCNCPoint5[17360] = {X 153.6431, Y 44.2084, Z -7.1667, A 0.000, B 0.000, C 0.000 }
gfCNCPoint5[17361] = {X 153.6429, Y 45.0400, Z -7.1667, A 0.000, B 0.000, C 0.000 }
gfCNCPoint5[17362] = {X 153.5310, Y 45.9591, Z -7.1667, A 0.000, B 0.000, C 0.000 }
gfCNCPoint5[17363] = {X 153.2186, Y 46.8306, Z -7.1667, A 0.000, B 0.000, C 0.000 }
gfCNCPoint5[17364] = {X 152.7212, Y 47.6115, Z -7.1667, A 0.000, B 0.000, C 0.000 }
gfCNCPoint5[17365] = {X 152.0634, Y 48.2631, Z -7.1667, A 0.000, B 0.000, C 0.000 }
gfCNCPoint5[17366] = {X 151.2778, Y 48.7530, Z -7.1667, A 0.000, B 0.000, C 0.000 }
gfCNCPoint5[17367] = {X 150.4032, Y 49.0570, Z -7.1667, A 0.000, B 0.000, C 0.000 }
gfCNCPoint5[17368] = {X 149.4831, Y 49.1600, Z -7.1667, A 0.000, B 0.000, C 0.000 }
gfCNCPoint5[17369] = {X 143.0396, Y 49.1600, Z -7.1667, A 0.000, B 0.000, C 0.000 }
gfCNCPoint5[17370] = {X 142.1185, Y 49.0567, Z -7.1667, A 0.000, B 0.000, C 0.000 }
gfCNCPoint5[17371] = {X 141.2432, Y 48.7521, Z -7.1667, A 0.000, B 0.000, C 0.000 }
gfCNCPoint5[17372] = {X 140.4570, Y 48.2612, Z -7.1667, A 0.000, B 0.000, C 0.000 }
gfCNCPoint5[17373] = {X 139.7990, Y 47.6084, Z -7.1667, A 0.000, B 0.000, C 0.000 }
gfCNCPoint5[17374] = {X 139.3019, Y 46.8261, Z -7.1667, A 0.000, B 0.000, C 0.000 }
gfCNCPoint5[17375] = {X 138.9903, Y 45.9532, Z -7.1667, A 0.000, B 0.000, C 0.000 }
gfCNCPoint5[17376] = {X 138.8798, Y 45.0329, Z -7.1667, A 0.000, B 0.000, C 0.000 }
gfCNCPoint5[17377] = {X 138.8800, Y 44.1516, Z -7.1667, A 0.000, B 0.000, C 0.000 }
gfCNCPoint5[17378] = {X 138.9906, Y 43.2545, Z -7.1667, A 0.000, B 0.000, C 0.000 }
gfCNCPoint5[17379] = {X 139.2922, Y 42.4026, Z -7.1667, A 0.000, B 0.000, C 0.000 }
gfCNCPoint5[17380] = {X 139.7708, Y 41.6358, Z -7.1667, A 0.000, B 0.000, C 0.000 }
gfCNCPoint5[17381] = {X 140.4036, Y 40.9906, Z -7.1667, A 0.000, B 0.000, C 0.000 }
gfCNCPoint5[17382] = {X 140.4036, Y 30.3969, Z -7.1667, A 0.000, B 0.000, C 0.000 }
gfCNCPoint5[17383] = {X 136.4036, Y 30.3969, Z -7.1667, A 0.000, B 0.000, C 0.000 }
gfCNCPoint5[17384] = {X 140.4836, Y 30.3969, Z -7.1667, A 0.000, B 0.000, C 0.000 }
gfCNCPoint5[17385] = {X 140.4836, Y 19.6382, Z -7.1667, A 0.000, B 0.000, C 0.000 }
gfCNCPoint5[17386] = {X 137.2911, Y 19.6379, Z -7.1667, A 0.000, B 0.000, C 0.000 }
gfCNCPoint5[17387] = {X 137.2218, Y 19.7475, Z -7.1667, A 0.000, B 0.000, C 0.000 }
gfCNCPoint5[17388] = {X 136.5756, Y 20.4907, Z -7.1667, A 0.000, B 0.000, C 0.000 }
gfCNCPoint5[17389] = {X 135.7702, Y 21.0573, Z -7.1667, A 0.000, B 0.000, C 0.000 }
gfCNCPoint5[17390] = {X 134.8524, Y 21.4145, Z -7.1667, A 0.000, B 0.000, C 0.000 }
gfCNCPoint5[17391] = {X 133.8758, Y 21.5414, Z -7.1667, A 0.000, B 0.000, C 0.000 }
gfCNCPoint5[17392] = {X 133.2006, Y 21.5415, Z -7.1667, A 0.000, B 0.000, C 0.000 }
gfCNCPoint5[17393] = {X 132.2928, Y 21.4392, Z -7.1667, A 0.000, B 0.000, C 0.000 }
gfCNCPoint5[17394] = {X 131.4304, Y 21.1375, Z -7.1667, A 0.000, B 0.000, C 0.000 }
gfCNCPoint5[17395] = {X 130.6568, Y 20.6514, Z -7.1667, A 0.000, B 0.000, C 0.000 }
gfCNCPoint5[17396] = {X 130.0108, Y 20.0054, Z -7.1667, A 0.000, B 0.000, C 0.000 }
gfCNCPoint5[17397] = {X 129.5247, Y 19.2318, Z -7.1667, A 0.000, B 0.000, C 0.000 }
gfCNCPoint5[17398] = {X 129.2229, Y 18.3694, Z -7.1667, A 0.000, B 0.000, C 0.000 }
gfCNCPoint5[17399] = {X 129.1206, Y 17.4615, Z -7.1667, A 0.000, B 0.000, C 0.000 }
gfCNCPoint5[17400] = {X 129.1206, Y 10.4835, Z -7.1667, A 0.000, B 0.000, C 0.000 }
gfCNCPoint5[17401] = {X 129.2215, Y 9.5820, Z -7.1667, A 0.000, B 0.000, C 0.000 }
gfCNCPoint5[17402] = {X 129.5191, Y 8.7250, Z -7.1667, A 0.000, B 0.000, C 0.000 }
gfCNCPoint5[17403] = {X 129.9986, Y 7.9550, Z -7.1667, A 0.000, B 0.000, C 0.000 }
gfCNCPoint5[17404] = {X 130.6365, Y 7.3099, Z -7.1667, A 0.000, B 0.000, C 0.000 }
gfCNCPoint5[17405] = {X 131.4011, Y 6.8218, Z -7.1667, A 0.000, B 0.000, C 0.000 }
gfCNCPoint5[17406] = {X 132.2547, Y 6.5147, Z -7.1667, A 0.000, B 0.000, C 0.000 }
gfCNCPoint5[17407] = {X 133.1551, Y 6.4038, Z -7.1667, A 0.000, B 0.000, C 0.000 }
gfCNCPoint5[17408] = {X 133.8841, Y 6.4037, Z -7.1667, A 0.000, B 0.000, C 0.000 }
gfCNCPoint5[17409] = {X 134.6871, Y 6.4919, Z -7.1667, A 0.000, B 0.000, C 0.000 }
gfCNCPoint5[17410] = {X 135.4570, Y 6.7366, Z -7.1667, A 0.000, B 0.000, C 0.000 }
gfCNCPoint5[17411] = {X 136.1635, Y 7.1282, Z -7.1667, A 0.000, B 0.000, C 0.000 }
gfCNCPoint5[17412] = {X 136.7791, Y 7.6512, Z -7.1667, A 0.000, B 0.000, C 0.000 }
gfCNCPoint5[17413] = {X 137.2795, Y 8.2854, Z -7.1667, A 0.000, B 0.000, C 0.000 }
gfCNCPoint5[17414] = {X 155.2423, Y 8.2867, Z -7.1667, A 0.000, B 0.000, C 0.000 }
gfCNCPoint5[17415] = {X 155.2878, Y 8.2171, Z -7.1667, A 0.000, B 0.000, C 0.000 }
gfCNCPoint5[17416] = {X 155.3347, Y 8.1485, Z -7.1667, A 0.000, B 0.000, C 0.000 }
gfCNCPoint5[17417] = {X 155.9798, Y 7.4252, Z -7.1667, A 0.000, B 0.000, C 0.000 }
gfCNCPoint5[17418] = {X 156.7773, Y 6.8746, Z -7.1667, A 0.000, B 0.000, C 0.000 }
gfCNCPoint5[17419] = {X 157.6822, Y 6.5275, Z -7.1667, A 0.000, B 0.000, C 0.000 }
gfCNCPoint5[17420] = {X 158.6434, Y 6.4037, Z -7.1667, A 0.000, B 0.000, C 0.000 }
gfCNCPoint5[17421] = {X 159.3750, Y 6.4039, Z -7.1667, A 0.000, B 0.000, C 0.000 }
gfCNCPoint5[17422] = {X 160.2741, Y 6.5161, Z -7.1667, A 0.000, B 0.000, C 0.000 }
gfCNCPoint5[17423] = {X 161.1263, Y 6.8241, Z -7.1667, A 0.000, B 0.000, C 0.000 }
gfCNCPoint5[17424] = {X 161.8895, Y 7.3126, Z -7.1667, A 0.000, B 0.000, C 0.000 }
gfCNCPoint5[17425] = {X 162.5260, Y 7.9574, Z -7.1667, A 0.000, B 0.000, C 0.000 }
gfCNCPoint5[17426] = {X 163.0046, Y 8.7269, Z -7.1667, A 0.000, B 0.000, C 0.000 }
gfCNCPoint5[17427] = {X 163.3015, Y 9.5830, Z -7.1667, A 0.000, B 0.000, C 0.000 }
gfCNCPoint5[17428] = {X 163.4021, Y 10.4835, Z -7.1667, A 0.000, B 0.000, C 0.000 }
gfCNCPoint5[17429] = {X 163.4021, Y 17.4615, Z -7.1667, A 0.000, B 0.000, C 0.000 }
gfCNCPoint5[17430] = {X 163.3015, Y 18.3621, Z -7.1667, A 0.000, B 0.000, C 0.000 }
gfCNCPoint5[17431] = {X 163.0046, Y 19.2182, Z -7.1667, A 0.000, B 0.000, C 0.000 }
gfCNCPoint5[17432] = {X 162.5260, Y 19.9876, Z -7.1667, A 0.000, B 0.000, C 0.000 }
gfCNCPoint5[17433] = {X 161.8895, Y 20.6325, Z -7.1667, A 0.000, B 0.000, C 0.000 }
gfCNCPoint5[17434] = {X 161.1263, Y 21.1209, Z -7.1667, A 0.000, B 0.000, C 0.000 }
gfCNCPoint5[17435] = {X 160.2741, Y 21.4289, Z -7.1667, A 0.000, B 0.000, C 0.000 }
gfCNCPoint5[17436] = {X 159.3750, Y 21.5412, Z -7.1667, A 0.000, B 0.000, C 0.000 }
gfCNCPoint5[17437] = {X 158.6802, Y 21.5415, Z -7.1667, A 0.000, B 0.000, C 0.000 }
gfCNCPoint5[17438] = {X 157.8634, Y 21.4567, Z -7.1667, A 0.000, B 0.000, C 0.000 }
gfCNCPoint5[17439] = {X 157.0797, Y 21.2112, Z -7.1667, A 0.000, B 0.000, C 0.000 }
gfCNCPoint5[17440] = {X 156.3605, Y 20.8147, Z -7.1667, A 0.000, B 0.000, C 0.000 }
gfCNCPoint5[17441] = {X 155.7345, Y 20.2832, Z -7.1667, A 0.000, B 0.000, C 0.000 }
gfCNCPoint5[17442] = {X 155.2267, Y 19.6379, Z -7.1667, A 0.000, B 0.000, C 0.000 }
gfCNCPoint5[17443] = {X 152.0372, Y 19.6389, Z -7.1667, A 0.000, B 0.000, C 0.000 }
gfCNCPoint5[17444] = {X 152.0361, Y 40.9684, Z -7.1667, A 0.000, B 0.000, C 0.000 }
gfCNCPoint5[17445] = {X 152.5609, Y 41.5335, Z -7.1667, A 0.000, B 0.000, C 0.000 }
gfCNCPoint5[17446] = {X 152.6515, Y 41.6413, Z -7.1667, A 0.000, B 0.000, C 0.000 }
gfCNCPoint5[17447] = {X 153.1474, Y 42.4206, Z -7.1667, A 0.000, B 0.000, C 0.000 }
gfCNCPoint5[17448] = {X 153.4565, Y 43.2911, Z -7.1667, A 0.000, B 0.000, C 0.000 }
gfCNCPoint5[17449] = {X 153.5631, Y 44.2086, Z -7.1667, A 0.000, B 0.000, C 0.000 }
gfCNCPoint5[17450] = {X 153.5629, Y 45.0392, Z -7.1667, A 0.000, B 0.000, C 0.000 }
gfCNCPoint5[17451] = {X 153.4532, Y 45.9406, Z -7.1667, A 0.000, B 0.000, C 0.000 }
gfCNCPoint5[17452] = {X 153.1468, Y 46.7954, Z -7.1667, A 0.000, B 0.000, C 0.000 }
gfCNCPoint5[17453] = {X 152.6589, Y 47.5613, Z -7.1667, A 0.000, B 0.000, C 0.000 }
gfCNCPoint5[17454] = {X 152.0138, Y 48.2003, Z -7.1667, A 0.000, B 0.000, C 0.000 }
gfCNCPoint5[17455] = {X 151.2432, Y 48.6808, Z -7.1667, A 0.000, B 0.000, C 0.000 }
gfCNCPoint5[17456] = {X 150.3855, Y 48.9789, Z -7.1667, A 0.000, B 0.000, C 0.000 }
gfCNCPoint5[17457] = {X 149.4831, Y 49.0800, Z -7.1667, A 0.000, B 0.000, C 0.000 }
gfCNCPoint5[17458] = {X 143.0396, Y 49.0800, Z -7.1667, A 0.000, B 0.000, C 0.000 }
gfCNCPoint5[17459] = {X 142.1362, Y 48.9787, Z -7.1667, A 0.000, B 0.000, C 0.000 }
gfCNCPoint5[17460] = {X 141.2777, Y 48.6799, Z -7.1667, A 0.000, B 0.000, C 0.000 }
gfCNCPoint5[17461] = {X 140.5066, Y 48.1985, Z -7.1667, A 0.000, B 0.000, C 0.000 }
gfCNCPoint5[17462] = {X 139.8613, Y 47.5582, Z -7.1667, A 0.000, B 0.000, C 0.000 }
gfCNCPoint5[17463] = {X 139.3737, Y 46.7910, Z -7.1667, A 0.000, B 0.000, C 0.000 }
gfCNCPoint5[17464] = {X 139.0682, Y 45.9349, Z -7.1667, A 0.000, B 0.000, C 0.000 }
gfCNCPoint5[17465] = {X 138.9598, Y 45.0323, Z -7.1667, A 0.000, B 0.000, C 0.000 }
gfCNCPoint5[17466] = {X 138.9600, Y 44.1527, Z -7.1667, A 0.000, B 0.000, C 0.000 }
gfCNCPoint5[17467] = {X 139.0706, Y 43.2637, Z -7.1667, A 0.000, B 0.000, C 0.000 }
gfCNCPoint5[17468] = {X 139.3725, Y 42.4203, Z -7.1667, A 0.000, B 0.000, C 0.000 }
gfCNCPoint5[17469] = {X 139.8512, Y 41.6631, Z -7.1667, A 0.000, B 0.000, C 0.000 }
gfCNCPoint5[17470] = {X 140.4836, Y 41.0287, Z -7.1667, A 0.000, B 0.000, C 0.000 }
gfCNCPoint5[17471] = {X 140.4836, Y 30.3969, Z -7.1667, A 0.000, B 0.000, C 0.000 }
gfCNCPoint5[17472] = {X 136.4836, Y 30.3969, Z -7.1667, A 0.000, B 0.000, C 0.000 }
gfCNCPoint5[17473] = {X 140.5636, Y 30.3969, Z -7.1667, A 0.000, B 0.000, C 0.000 }
gfCNCPoint5[17474] = {X 140.5636, Y 19.5583, Z -7.1667, A 0.000, B 0.000, C 0.000 }
gfCNCPoint5[17475] = {X 137.2663, Y 19.5579, Z -7.1667, A 0.000, B 0.000, C 0.000 }
gfCNCPoint5[17476] = {X 137.2445, Y 19.5618, Z -7.1667, A 0.000, B 0.000, C 0.000 }
gfCNCPoint5[17477] = {X 137.1362, Y 19.7309, Z -7.1667, A 0.000, B 0.000, C 0.000 }
gfCNCPoint5[17478] = {X 136.4967, Y 20.4539, Z -7.1667, A 0.000, B 0.000, C 0.000 }
gfCNCPoint5[17479] = {X 135.7027, Y 21.0026, Z -7.1667, A 0.000, B 0.000, C 0.000 }
gfCNCPoint5[17480] = {X 134.8003, Y 21.3451, Z -7.1667, A 0.000, B 0.000, C 0.000 }
gfCNCPoint5[17481] = {X 133.8422, Y 21.4615, Z -7.1667, A 0.000, B 0.000, C 0.000 }
gfCNCPoint5[17482] = {X 133.2006, Y 21.4615, Z -7.1667, A 0.000, B 0.000, C 0.000 }
gfCNCPoint5[17483] = {X 132.3106, Y 21.3612, Z -7.1667, A 0.000, B 0.000, C 0.000 }
gfCNCPoint5[17484] = {X 131.4651, Y 21.0654, Z -7.1667, A 0.000, B 0.000, C 0.000 }
gfCNCPoint5[17485] = {X 130.7067, Y 20.5889, Z -7.1667, A 0.000, B 0.000, C 0.000 }
gfCNCPoint5[17486] = {X 130.0733, Y 19.9555, Z -7.1667, A 0.000, B 0.000, C 0.000 }
gfCNCPoint5[17487] = {X 129.5968, Y 19.1971, Z -7.1667, A 0.000, B 0.000, C 0.000 }
gfCNCPoint5[17488] = {X 129.3009, Y 18.3516, Z -7.1667, A 0.000, B 0.000, C 0.000 }
gfCNCPoint5[17489] = {X 129.2006, Y 17.4615, Z -7.1667, A 0.000, B 0.000, C 0.000 }
gfCNCPoint5[17490] = {X 129.2006, Y 10.4835, Z -7.1667, A 0.000, B 0.000, C 0.000 }
gfCNCPoint5[17491] = {X 129.3009, Y 9.5934, Z -7.1667, A 0.000, B 0.000, C 0.000 }
gfCNCPoint5[17492] = {X 129.5968, Y 8.7480, Z -7.1667, A 0.000, B 0.000, C 0.000 }
gfCNCPoint5[17493] = {X 130.0733, Y 7.9896, Z -7.1667, A 0.000, B 0.000, C 0.000 }
gfCNCPoint5[17494] = {X 130.7067, Y 7.3562, Z -7.1667, A 0.000, B 0.000, C 0.000 }
gfCNCPoint5[17495] = {X 131.4651, Y 6.8796, Z -7.1667, A 0.000, B 0.000, C 0.000 }
gfCNCPoint5[17496] = {X 132.3106, Y 6.5838, Z -7.1667, A 0.000, B 0.000, C 0.000 }
gfCNCPoint5[17497] = {X 133.2007, Y 6.4835, Z -7.1667, A 0.000, B 0.000, C 0.000 }
gfCNCPoint5[17498] = {X 133.8833, Y 6.4837, Z -7.1667, A 0.000, B 0.000, C 0.000 }
gfCNCPoint5[17499] = {X 134.6791, Y 6.5720, Z -7.1667, A 0.000, B 0.000, C 0.000 }
gfCNCPoint5[17500] = {X 135.4413, Y 6.8170, Z -7.1667, A 0.000, B 0.000, C 0.000 }
gfCNCPoint5[17501] = {X 136.1395, Y 7.2089, Z -7.1667, A 0.000, B 0.000, C 0.000 }
gfCNCPoint5[17502] = {X 136.7456, Y 7.7320, Z -7.1667, A 0.000, B 0.000, C 0.000 }
gfCNCPoint5[17503] = {X 137.2355, Y 8.3654, Z -7.1667, A 0.000, B 0.000, C 0.000 }
gfCNCPoint5[17504] = {X 155.2276, Y 8.3654, Z -7.1667, A 0.000, B 0.000, C 0.000 }
gfCNCPoint5[17505] = {X 155.2814, Y 8.3748, Z -7.1667, A 0.000, B 0.000, C 0.000 }
gfCNCPoint5[17506] = {X 155.3396, Y 8.2837, Z -7.1667, A 0.000, B 0.000, C 0.000 }
gfCNCPoint5[17507] = {X 155.4003, Y 8.1943, Z -7.1667, A 0.000, B 0.000, C 0.000 }
gfCNCPoint5[17508] = {X 156.0396, Y 7.4792, Z -7.1667, A 0.000, B 0.000, C 0.000 }
gfCNCPoint5[17509] = {X 156.8307, Y 6.9369, Z -7.1667, A 0.000, B 0.000, C 0.000 }
gfCNCPoint5[17510] = {X 157.7283, Y 6.5985, Z -7.1667, A 0.000, B 0.000, C 0.000 }
gfCNCPoint5[17511] = {X 158.6805, Y 6.4835, Z -7.1667, A 0.000, B 0.000, C 0.000 }
gfCNCPoint5[17512] = {X 159.3739, Y 6.4839, Z -7.1667, A 0.000, B 0.000, C 0.000 }
gfCNCPoint5[17513] = {X 160.2554, Y 6.5939, Z -7.1667, A 0.000, B 0.000, C 0.000 }
gfCNCPoint5[17514] = {X 161.0909, Y 6.8959, Z -7.1667, A 0.000, B 0.000, C 0.000 }
gfCNCPoint5[17515] = {X 161.8391, Y 7.3747, Z -7.1667, A 0.000, B 0.000, C 0.000 }
gfCNCPoint5[17516] = {X 162.4632, Y 8.0070, Z -7.1667, A 0.000, B 0.000, C 0.000 }
gfCNCPoint5[17517] = {X 162.9324, Y 8.7613, Z -7.1667, A 0.000, B 0.000, C 0.000 }
gfCNCPoint5[17518] = {X 163.2234, Y 9.6007, Z -7.1667, A 0.000, B 0.000, C 0.000 }
gfCNCPoint5[17519] = {X 163.3221, Y 10.4835, Z -7.1667, A 0.000, B 0.000, C 0.000 }
gfCNCPoint5[17520] = {X 163.3221, Y 17.4615, Z -7.1667, A 0.000, B 0.000, C 0.000 }
gfCNCPoint5[17521] = {X 163.2218, Y 18.3516, Z -7.1667, A 0.000, B 0.000, C 0.000 }
gfCNCPoint5[17522] = {X 162.9260, Y 19.1971, Z -7.1667, A 0.000, B 0.000, C 0.000 }
gfCNCPoint5[17523] = {X 162.4494, Y 19.9555, Z -7.1667, A 0.000, B 0.000, C 0.000 }
gfCNCPoint5[17524] = {X 161.8160, Y 20.5889, Z -7.1667, A 0.000, B 0.000, C 0.000 }
gfCNCPoint5[17525] = {X 161.0576, Y 21.0654, Z -7.1667, A 0.000, B 0.000, C 0.000 }
gfCNCPoint5[17526] = {X 160.2122, Y 21.3613, Z -7.1667, A 0.000, B 0.000, C 0.000 }
gfCNCPoint5[17527] = {X 159.3221, Y 21.4615, Z -7.1667, A 0.000, B 0.000, C 0.000 }
gfCNCPoint5[17528] = {X 158.6805, Y 21.4615, Z -7.1667, A 0.000, B 0.000, C 0.000 }
gfCNCPoint5[17529] = {X 157.8710, Y 21.3766, Z -7.1667, A 0.000, B 0.000, C 0.000 }
gfCNCPoint5[17530] = {X 157.0951, Y 21.1307, Z -7.1667, A 0.000, B 0.000, C 0.000 }
gfCNCPoint5[17531] = {X 156.3844, Y 20.7339, Z -7.1667, A 0.000, B 0.000, C 0.000 }
gfCNCPoint5[17532] = {X 155.7679, Y 20.2024, Z -7.1667, A 0.000, B 0.000, C 0.000 }
gfCNCPoint5[17533] = {X 155.2709, Y 19.5579, Z -7.1667, A 0.000, B 0.000, C 0.000 }
gfCNCPoint5[17534] = {X 151.9572, Y 19.5590, Z -7.1667, A 0.000, B 0.000, C 0.000 }
gfCNCPoint5[17535] = {X 151.9561, Y 40.9999, Z -7.1667, A 0.000, B 0.000, C 0.000 }
gfCNCPoint5[17536] = {X 152.5009, Y 41.5865, Z -7.1667, A 0.000, B 0.000, C 0.000 }
gfCNCPoint5[17537] = {X 152.5898, Y 41.6922, Z -7.1667, A 0.000, B 0.000, C 0.000 }
gfCNCPoint5[17538] = {X 153.0757, Y 42.4562, Z -7.1667, A 0.000, B 0.000, C 0.000 }
gfCNCPoint5[17539] = {X 153.3786, Y 43.3095, Z -7.1667, A 0.000, B 0.000, C 0.000 }
gfCNCPoint5[17540] = {X 153.4831, Y 44.2088, Z -7.1667, A 0.000, B 0.000, C 0.000 }
gfCNCPoint5[17541] = {X 153.4829, Y 45.0384, Z -7.1667, A 0.000, B 0.000, C 0.000 }
gfCNCPoint5[17542] = {X 153.3753, Y 45.9222, Z -7.1667, A 0.000, B 0.000, C 0.000 }
gfCNCPoint5[17543] = {X 153.0750, Y 46.7602, Z -7.1667, A 0.000, B 0.000, C 0.000 }
gfCNCPoint5[17544] = {X 152.5967, Y 47.5111, Z -7.1667, A 0.000, B 0.000, C 0.000 }
gfCNCPoint5[17545] = {X 151.9642, Y 48.1376, Z -7.1667, A 0.000, B 0.000, C 0.000 }
gfCNCPoint5[17546] = {X 151.2087, Y 48.6086, Z -7.1667, A 0.000, B 0.000, C 0.000 }
gfCNCPoint5[17547] = {X 150.3678, Y 48.9009, Z -7.1667, A 0.000, B 0.000, C 0.000 }
gfCNCPoint5[17548] = {X 149.4831, Y 49.0000, Z -7.1667, A 0.000, B 0.000, C 0.000 }
gfCNCPoint5[17549] = {X 143.0396, Y 49.0000, Z -7.1667, A 0.000, B 0.000, C 0.000 }
gfCNCPoint5[17550] = {X 142.1495, Y 48.8997, Z -7.1667, A 0.000, B 0.000, C 0.000 }
gfCNCPoint5[17551] = {X 141.3041, Y 48.6039, Z -7.1667, A 0.000, B 0.000, C 0.000 }
gfCNCPoint5[17552] = {X 140.5457, Y 48.1273, Z -7.1667, A 0.000, B 0.000, C 0.000 }
gfCNCPoint5[17553] = {X 139.9123, Y 47.4939, Z -7.1667, A 0.000, B 0.000, C 0.000 }
gfCNCPoint5[17554] = {X 139.4357, Y 46.7355, Z -7.1667, A 0.000, B 0.000, C 0.000 }
gfCNCPoint5[17555] = {X 139.1399, Y 45.8901, Z -7.1667, A 0.000, B 0.000, C 0.000 }
gfCNCPoint5[17556] = {X 139.0396, Y 45.0000, Z -7.1667, A 0.000, B 0.000, C 0.000 }
gfCNCPoint5[17557] = {X 139.0400, Y 44.1538, Z -7.1667, A 0.000, B 0.000, C 0.000 }
gfCNCPoint5[17558] = {X 139.1506, Y 43.2730, Z -7.1667, A 0.000, B 0.000, C 0.000 }
gfCNCPoint5[17559] = {X 139.4528, Y 42.4382, Z -7.1667, A 0.000, B 0.000, C 0.000 }
gfCNCPoint5[17560] = {X 139.9317, Y 41.6907, Z -7.1667, A 0.000, B 0.000, C 0.000 }
gfCNCPoint5[17561] = {X 140.5636, Y 41.0672, Z -7.1667, A 0.000, B 0.000, C 0.000 }
gfCNCPoint5[17562] = {X 140.5636, Y 30.3969, Z -7.1667, A 0.000, B 0.000, C 0.000 }
gfCNCPoint5[17563] = {X 136.4836, Y 30.3969, Z -7.1667, A 0.000, B 0.000, C 0.000 }
gfCNCPoint5[17564] = {X 136.4836, Y 30.3969, Z -4.1667, A 0.000, B 0.000, C 0.000 }
gfCNCPoint5[17565] = {X 136.4836, Y 30.3969, Z 11.0000, A 0.000, B 0.000, C 0.000 }
gfCNCPoint5[17566] = {X 137.6628, Y 74.8913, Z 11.0000, A 0.000, B 0.000, C 0.000 }
gfCNCPoint5[17567] = {X 137.6628, Y 74.8913, Z -4.1667, A 0.000, B 0.000, C 0.000 }
gfCNCPoint5[17568] = {X 137.6628, Y 74.8913, Z -7.1667, A 0.000, B 0.000, C 0.000 }
gfCNCPoint5[17569] = {X 140.6794, Y 77.6384, Z -7.1667, A 0.000, B 0.000, C 0.000 }
gfCNCPoint5[17570] = {X 155.6320, Y 61.2195, Z -7.1667, A 0.000, B 0.000, C 0.000 }
gfCNCPoint5[17571] = {X 155.2772, Y 60.5139, Z -7.1667, A 0.000, B 0.000, C 0.000 }
gfCNCPoint5[17572] = {X 155.0568, Y 59.7555, Z -7.1667, A 0.000, B 0.000, C 0.000 }
gfCNCPoint5[17573] = {X 154.9781, Y 58.9697, Z -7.1667, A 0.000, B 0.000, C 0.000 }
gfCNCPoint5[17574] = {X 154.9780, Y 58.0000, Z -7.1667, A 0.000, B 0.000, C 0.000 }
gfCNCPoint5[17575] = {X 155.0863, Y 57.0387, Z -7.1667, A 0.000, B 0.000, C 0.000 }
gfCNCPoint5[17576] = {X 155.4058, Y 56.1256, Z -7.1667, A 0.000, B 0.000, C 0.000 }
gfCNCPoint5[17577] = {X 155.9204, Y 55.3065, Z -7.1667, A 0.000, B 0.000, C 0.000 }
gfCNCPoint5[17578] = {X 156.6045, Y 54.6225, Z -7.1667, A 0.000, B 0.000, C 0.000 }
gfCNCPoint5[17579] = {X 157.4236, Y 54.1078, Z -7.1667, A 0.000, B 0.000, C 0.000 }
gfCNCPoint5[17580] = {X 158.3367, Y 53.7883, Z -7.1667, A 0.000, B 0.000, C 0.000 }
gfCNCPoint5[17581] = {X 159.2980, Y 53.6800, Z -7.1667, A 0.000, B 0.000, C 0.000 }
gfCNCPoint5[17582] = {X 178.5335, Y 53.6800, Z -7.1667, A 0.000, B 0.000, C 0.000 }
gfCNCPoint5[17583] = {X 179.4948, Y 53.7883, Z -7.1667, A 0.000, B 0.000, C 0.000 }
gfCNCPoint5[17584] = {X 180.4079, Y 54.1078, Z -7.1667, A 0.000, B 0.000, C 0.000 }
gfCNCPoint5[17585] = {X 181.2270, Y 54.6225, Z -7.1667, A 0.000, B 0.000, C 0.000 }
gfCNCPoint5[17586] = {X 181.9110, Y 55.3065, Z -7.1667, A 0.000, B 0.000, C 0.000 }
gfCNCPoint5[17587] = {X 182.4257, Y 56.1256, Z -7.1667, A 0.000, B 0.000, C 0.000 }
gfCNCPoint5[17588] = {X 182.7452, Y 57.0387, Z -7.1667, A 0.000, B 0.000, C 0.000 }
gfCNCPoint5[17589] = {X 182.8535, Y 58.0000, Z -7.1667, A 0.000, B 0.000, C 0.000 }
gfCNCPoint5[17590] = {X 182.8535, Y 58.9342, Z -7.1667, A 0.000, B 0.000, C 0.000 }
gfCNCPoint5[17591] = {X 182.7808, Y 59.7230, Z -7.1667, A 0.000, B 0.000, C 0.000 }
gfCNCPoint5[17592] = {X 182.5654, Y 60.4853, Z -7.1667, A 0.000, B 0.000, C 0.000 }
gfCNCPoint5[17593] = {X 182.2144, Y 61.1954, Z -7.1667, A 0.000, B 0.000, C 0.000 }
gfCNCPoint5[17594] = {X 209.2964, Y 90.7596, Z -7.1667, A 0.000, B 0.000, C 0.000 }
gfCNCPoint5[17595] = {X 209.9675, Y 91.4547, Z -7.1667, A 0.000, B 0.000, C 0.000 }
gfCNCPoint5[17596] = {X 210.6741, Y 92.1135, Z -7.1667, A 0.000, B 0.000, C 0.000 }
gfCNCPoint5[17597] = {X 211.0673, Y 92.3796, Z -7.1667, A 0.000, B 0.000, C 0.000 }
gfCNCPoint5[17598] = {X 211.5153, Y 92.5364, Z -7.1667, A 0.000, B 0.000, C 0.000 }
gfCNCPoint5[17599] = {X 212.1076, Y 92.6610, Z -7.1667, A 0.000, B 0.000, C 0.000 }
gfCNCPoint5[17600] = {X 213.3747, Y 92.8206, Z -7.1667, A 0.000, B 0.000, C 0.000 }
gfCNCPoint5[17601] = {X 214.4399, Y 92.7363, Z -7.1667, A 0.000, B 0.000, C 0.000 }
gfCNCPoint5[17602] = {X 215.5067, Y 92.6746, Z -7.1667, A 0.000, B 0.000, C 0.000 }
gfCNCPoint5[17603] = {X 216.1770, Y 92.6016, Z -7.1667, A 0.000, B 0.000, C 0.000 }
gfCNCPoint5[17604] = {X 216.8224, Y 92.4066, Z -7.1667, A 0.000, B 0.000, C 0.000 }
gfCNCPoint5[17605] = {X 217.4209, Y 92.0961, Z -7.1667, A 0.000, B 0.000, C 0.000 }
gfCNCPoint5[17606] = {X 222.9613, Y 88.5206, Z -7.1667, A 0.000, B 0.000, C 0.000 }
gfCNCPoint5[17607] = {X 245.8271, Y 73.8997, Z -7.1667, A 0.000, B 0.000, C 0.000 }
gfCNCPoint5[17608] = {X 221.6306, Y 64.4047, Z -7.1667, A 0.000, B 0.000, C 0.000 }
gfCNCPoint5[17609] = {X 219.8631, Y 63.8132, Z -7.1667, A 0.000, B 0.000, C 0.000 }
gfCNCPoint5[17610] = {X 218.0397, Y 63.4272, Z -7.1667, A 0.000, B 0.000, C 0.000 }
gfCNCPoint5[17611] = {X 216.1841, Y 63.2516, Z -7.1667, A 0.000, B 0.000, C 0.000 }
gfCNCPoint5[17612] = {X 215.2522, Y 63.1173, Z -7.1667, A 0.000, B 0.000, C 0.000 }
gfCNCPoint5[17613] = {X 214.3716, Y 62.7843, Z -7.1667, A 0.000, B 0.000, C 0.000 }
gfCNCPoint5[17614] = {X 213.5841, Y 62.2684, Z -7.1667, A 0.000, B 0.000, C 0.000 }
gfCNCPoint5[17615] = {X 212.9270, Y 61.5942, Z -7.1667, A 0.000, B 0.000, C 0.000 }
gfCNCPoint5[17616] = {X 212.4315, Y 60.7936, Z -7.1667, A 0.000, B 0.000, C 0.000 }
gfCNCPoint5[17617] = {X 212.1213, Y 59.9047, Z -7.1667, A 0.000, B 0.000, C 0.000 }
gfCNCPoint5[17618] = {X 212.0110, Y 58.9697, Z -7.1667, A 0.000, B 0.000, C 0.000 }
gfCNCPoint5[17619] = {X 212.0108, Y 58.0000, Z -7.1667, A 0.000, B 0.000, C 0.000 }
gfCNCPoint5[17620] = {X 212.1191, Y 57.0387, Z -7.1667, A 0.000, B 0.000, C 0.000 }
gfCNCPoint5[17621] = {X 212.4386, Y 56.1256, Z -7.1667, A 0.000, B 0.000, C 0.000 }
gfCNCPoint5[17622] = {X 212.9533, Y 55.3065, Z -7.1667, A 0.000, B 0.000, C 0.000 }
gfCNCPoint5[17623] = {X 213.6373, Y 54.6225, Z -7.1667, A 0.000, B 0.000, C 0.000 }
gfCNCPoint5[17624] = {X 214.4564, Y 54.1078, Z -7.1667, A 0.000, B 0.000, C 0.000 }
gfCNCPoint5[17625] = {X 215.3695, Y 53.7883, Z -7.1667, A 0.000, B 0.000, C 0.000 }
gfCNCPoint5[17626] = {X 216.3308, Y 53.6800, Z -7.1667, A 0.000, B 0.000, C 0.000 }
gfCNCPoint5[17627] = {X 237.2617, Y 53.6800, Z -7.1667, A 0.000, B 0.000, C 0.000 }
gfCNCPoint5[17628] = {X 238.2230, Y 53.7883, Z -7.1667, A 0.000, B 0.000, C 0.000 }
gfCNCPoint5[17629] = {X 239.1361, Y 54.1078, Z -7.1667, A 0.000, B 0.000, C 0.000 }
gfCNCPoint5[17630] = {X 239.9552, Y 54.6225, Z -7.1667, A 0.000, B 0.000, C 0.000 }
gfCNCPoint5[17631] = {X 240.6392, Y 55.3065, Z -7.1667, A 0.000, B 0.000, C 0.000 }
gfCNCPoint5[17632] = {X 241.1539, Y 56.1256, Z -7.1667, A 0.000, B 0.000, C 0.000 }
gfCNCPoint5[17633] = {X 241.4734, Y 57.0387, Z -7.1667, A 0.000, B 0.000, C 0.000 }
gfCNCPoint5[17634] = {X 241.5817, Y 58.0000, Z -7.1667, A 0.000, B 0.000, C 0.000 }
gfCNCPoint5[17635] = {X 241.5817, Y 58.2317, Z -7.1667, A 0.000, B 0.000, C 0.000 }
gfCNCPoint5[17636] = {X 248.1148, Y 60.7793, Z -7.1667, A 0.000, B 0.000, C 0.000 }
gfCNCPoint5[17637] = {X 275.6319, Y 71.7013, Z -7.1667, A 0.000, B 0.000, C 0.000 }
gfCNCPoint5[17638] = {X 275.6335, Y 63.2123, Z -7.1667, A 0.000, B 0.000, C 0.000 }
gfCNCPoint5[17639] = {X 274.7819, Y 63.0032, Z -7.1667, A 0.000, B 0.000, C 0.000 }
gfCNCPoint5[17640] = {X 273.9900, Y 62.6263, Z -7.1667, A 0.000, B 0.000, C 0.000 }
gfCNCPoint5[17641] = {X 273.2906, Y 62.0974, Z -7.1667, A 0.000, B 0.000, C 0.000 }
gfCNCPoint5[17642] = {X 272.7124, Y 61.4381, Z -7.1667, A 0.000, B 0.000, C 0.000 }
gfCNCPoint5[17643] = {X 272.2793, Y 60.6756, Z -7.1667, A 0.000, B 0.000, C 0.000 }
gfCNCPoint5[17644] = {X 272.0090, Y 59.8414, Z -7.1667, A 0.000, B 0.000, C 0.000 }
gfCNCPoint5[17645] = {X 271.9128, Y 58.9697, Z -7.1667, A 0.000, B 0.000, C 0.000 }
gfCNCPoint5[17646] = {X 271.9127, Y 58.0000, Z -7.1667, A 0.000, B 0.000, C 0.000 }
gfCNCPoint5[17647] = {X 272.0210, Y 57.0387, Z -7.1667, A 0.000, B 0.000, C 0.000 }
gfCNCPoint5[17648] = {X 272.3405, Y 56.1256, Z -7.1667, A 0.000, B 0.000, C 0.000 }
gfCNCPoint5[17649] = {X 272.8552, Y 55.3065, Z -7.1667, A 0.000, B 0.000, C 0.000 }
gfCNCPoint5[17650] = {X 273.5392, Y 54.6225, Z -7.1667, A 0.000, B 0.000, C 0.000 }
gfCNCPoint5[17651] = {X 274.3583, Y 54.1078, Z -7.1667, A 0.000, B 0.000, C 0.000 }
gfCNCPoint5[17652] = {X 275.2714, Y 53.7883, Z -7.1667, A 0.000, B 0.000, C 0.000 }
gfCNCPoint5[17653] = {X 276.2327, Y 53.6800, Z -7.1667, A 0.000, B 0.000, C 0.000 }
gfCNCPoint5[17654] = {X 292.7731, Y 53.6800, Z -7.1667, A 0.000, B 0.000, C 0.000 }
gfCNCPoint5[17655] = {X 293.7344, Y 53.7883, Z -7.1667, A 0.000, B 0.000, C 0.000 }
gfCNCPoint5[17656] = {X 294.6475, Y 54.1078, Z -7.1667, A 0.000, B 0.000, C 0.000 }
gfCNCPoint5[17657] = {X 295.4666, Y 54.6225, Z -7.1667, A 0.000, B 0.000, C 0.000 }
gfCNCPoint5[17658] = {X 296.1506, Y 55.3065, Z -7.1667, A 0.000, B 0.000, C 0.000 }
gfCNCPoint5[17659] = {X 296.6653, Y 56.1256, Z -7.1667, A 0.000, B 0.000, C 0.000 }
gfCNCPoint5[17660] = {X 296.9848, Y 57.0387, Z -7.1667, A 0.000, B 0.000, C 0.000 }
gfCNCPoint5[17661] = {X 297.0931, Y 58.0000, Z -7.1667, A 0.000, B 0.000, C 0.000 }
gfCNCPoint5[17662] = {X 297.0931, Y 58.9350, Z -7.1667, A 0.000, B 0.000, C 0.000 }
gfCNCPoint5[17663] = {X 297.0011, Y 59.8115, Z -7.1667, A 0.000, B 0.000, C 0.000 }
gfCNCPoint5[17664] = {X 296.7337, Y 60.6514, Z -7.1667, A 0.000, B 0.000, C 0.000 }
gfCNCPoint5[17665] = {X 296.3021, Y 61.4198, Z -7.1667, A 0.000, B 0.000, C 0.000 }
gfCNCPoint5[17666] = {X 295.7240, Y 62.0851, Z -7.1667, A 0.000, B 0.000, C 0.000 }
gfCNCPoint5[17667] = {X 295.0233, Y 62.6197, Z -7.1667, A 0.000, B 0.000, C 0.000 }
gfCNCPoint5[17668] = {X 294.2289, Y 63.0016, Z -7.1667, A 0.000, B 0.000, C 0.000 }
gfCNCPoint5[17669] = {X 293.3738, Y 63.2150, Z -7.1667, A 0.000, B 0.000, C 0.000 }
gfCNCPoint5[17670] = {X 293.3849, Y 92.7802, Z -7.1667, A 0.000, B 0.000, C 0.000 }
gfCNCPoint5[17671] = {X 294.2375, Y 92.9977, Z -7.1667, A 0.000, B 0.000, C 0.000 }
gfCNCPoint5[17672] = {X 295.0289, Y 93.3823, Z -7.1667, A 0.000, B 0.000, C 0.000 }
gfCNCPoint5[17673] = {X 295.7269, Y 93.9182, Z -7.1667, A 0.000, B 0.000, C 0.000 }
gfCNCPoint5[17674] = {X 296.3027, Y 94.5835, Z -7.1667, A 0.000, B 0.000, C 0.000 }
gfCNCPoint5[17675] = {X 296.7330, Y 95.3511, Z -7.1667, A 0.000, B 0.000, C 0.000 }
gfCNCPoint5[17676] = {X 297.0001, Y 96.1895, Z -7.1667, A 0.000, B 0.000, C 0.000 }
gfCNCPoint5[17677] = {X 297.0931, Y 97.0645, Z -7.1667, A 0.000, B 0.000, C 0.000 }
gfCNCPoint5[17678] = {X 297.0931, Y 98.0000, Z -7.1667, A 0.000, B 0.000, C 0.000 }
gfCNCPoint5[17679] = {X 296.9848, Y 98.9613, Z -7.1667, A 0.000, B 0.000, C 0.000 }
gfCNCPoint5[17680] = {X 296.6653, Y 99.8744, Z -7.1667, A 0.000, B 0.000, C 0.000 }
gfCNCPoint5[17681] = {X 296.1506, Y 100.6935, Z -7.1667, A 0.000, B 0.000, C 0.000 }
gfCNCPoint5[17682] = {X 295.4666, Y 101.3775, Z -7.1667, A 0.000, B 0.000, C 0.000 }
gfCNCPoint5[17683] = {X 294.6475, Y 101.8922, Z -7.1667, A 0.000, B 0.000, C 0.000 }
gfCNCPoint5[17684] = {X 293.7344, Y 102.2117, Z -7.1667, A 0.000, B 0.000, C 0.000 }
gfCNCPoint5[17685] = {X 292.7731, Y 102.3200, Z -7.1667, A 0.000, B 0.000, C 0.000 }
gfCNCPoint5[17686] = {X 276.2327, Y 102.3200, Z -7.1667, A 0.000, B 0.000, C 0.000 }
gfCNCPoint5[17687] = {X 275.2714, Y 102.2117, Z -7.1667, A 0.000, B 0.000, C 0.000 }
gfCNCPoint5[17688] = {X 274.3583, Y 101.8922, Z -7.1667, A 0.000, B 0.000, C 0.000 }
gfCNCPoint5[17689] = {X 273.5392, Y 101.3775, Z -7.1667, A 0.000, B 0.000, C 0.000 }
gfCNCPoint5[17690] = {X 272.8552, Y 100.6935, Z -7.1667, A 0.000, B 0.000, C 0.000 }
gfCNCPoint5[17691] = {X 272.3405, Y 99.8744, Z -7.1667, A 0.000, B 0.000, C 0.000 }
gfCNCPoint5[17692] = {X 272.0210, Y 98.9613, Z -7.1667, A 0.000, B 0.000, C 0.000 }
gfCNCPoint5[17693] = {X 271.9127, Y 98.0000, Z -7.1667, A 0.000, B 0.000, C 0.000 }
gfCNCPoint5[17694] = {X 271.9127, Y 97.0658, Z -7.1667, A 0.000, B 0.000, C 0.000 }
gfCNCPoint5[17695] = {X 272.0026, Y 96.1890, Z -7.1667, A 0.000, B 0.000, C 0.000 }
gfCNCPoint5[17696] = {X 272.2686, Y 95.3488, Z -7.1667, A 0.000, B 0.000, C 0.000 }
gfCNCPoint5[17697] = {X 272.6997, Y 94.5800, Z -7.1667, A 0.000, B 0.000, C 0.000 }
gfCNCPoint5[17698] = {X 273.2777, Y 93.9146, Z -7.1667, A 0.000, B 0.000, C 0.000 }
gfCNCPoint5[17699] = {X 273.9788, Y 93.3805, Z -7.1667, A 0.000, B 0.000, C 0.000 }
gfCNCPoint5[17700] = {X 274.7737, Y 92.9997, Z -7.1667, A 0.000, B 0.000, C 0.000 }
gfCNCPoint5[17701] = {X 275.6294, Y 92.7883, Z -7.1667, A 0.000, B 0.000, C 0.000 }
gfCNCPoint5[17702] = {X 275.6294, Y 85.5950, Z -7.1667, A 0.000, B 0.000, C 0.000 }
gfCNCPoint5[17703] = {X 262.6399, Y 80.5031, Z -7.1667, A 0.000, B 0.000, C 0.000 }
gfCNCPoint5[17704] = {X 262.2782, Y 80.7315, Z -7.1667, A 0.000, B 0.000, C 0.000 }
gfCNCPoint5[17705] = {X 237.7974, Y 96.5884, Z -7.1667, A 0.000, B 0.000, C 0.000 }
gfCNCPoint5[17706] = {X 237.7998, Y 97.0651, Z -7.1667, A 0.000, B 0.000, C 0.000 }
gfCNCPoint5[17707] = {X 237.7998, Y 98.0000, Z -7.1667, A 0.000, B 0.000, C 0.000 }
gfCNCPoint5[17708] = {X 237.6915, Y 98.9613, Z -7.1667, A 0.000, B 0.000, C 0.000 }
gfCNCPoint5[17709] = {X 237.3720, Y 99.8744, Z -7.1667, A 0.000, B 0.000, C 0.000 }
gfCNCPoint5[17710] = {X 236.8573, Y 100.6935, Z -7.1667, A 0.000, B 0.000, C 0.000 }
gfCNCPoint5[17711] = {X 236.1733, Y 101.3775, Z -7.1667, A 0.000, B 0.000, C 0.000 }
gfCNCPoint5[17712] = {X 235.3542, Y 101.8922, Z -7.1667, A 0.000, B 0.000, C 0.000 }
gfCNCPoint5[17713] = {X 234.4411, Y 102.2117, Z -7.1667, A 0.000, B 0.000, C 0.000 }
gfCNCPoint5[17714] = {X 233.4798, Y 102.3200, Z -7.1667, A 0.000, B 0.000, C 0.000 }
gfCNCPoint5[17715] = {X 214.1790, Y 102.3200, Z -7.1667, A 0.000, B 0.000, C 0.000 }
gfCNCPoint5[17716] = {X 213.7862, Y 102.3021, Z -7.1667, A 0.000, B 0.000, C 0.000 }
gfCNCPoint5[17717] = {X 213.3966, Y 102.2485, Z -7.1667, A 0.000, B 0.000, C 0.000 }
gfCNCPoint5[17718] = {X 213.0070, Y 102.3021, Z -7.1667, A 0.000, B 0.000, C 0.000 }
gfCNCPoint5[17719] = {X 212.6141, Y 102.3200, Z -7.1667, A 0.000, B 0.000, C 0.000 }
gfCNCPoint5[17720] = {X 194.9870, Y 102.3200, Z -7.1667, A 0.000, B 0.000, C 0.000 }
gfCNCPoint5[17721] = {X 194.0257, Y 102.2117, Z -7.1667, A 0.000, B 0.000, C 0.000 }
gfCNCPoint5[17722] = {X 193.1126, Y 101.8922, Z -7.1667, A 0.000, B 0.000, C 0.000 }
gfCNCPoint5[17723] = {X 192.2935, Y 101.3775, Z -7.1667, A 0.000, B 0.000, C 0.000 }
gfCNCPoint5[17724] = {X 191.6094, Y 100.6935, Z -7.1667, A 0.000, B 0.000, C 0.000 }
gfCNCPoint5[17725] = {X 191.0948, Y 99.8744, Z -7.1667, A 0.000, B 0.000, C 0.000 }
gfCNCPoint5[17726] = {X 190.7753, Y 98.9613, Z -7.1667, A 0.000, B 0.000, C 0.000 }
gfCNCPoint5[17727] = {X 190.6670, Y 98.0000, Z -7.1667, A 0.000, B 0.000, C 0.000 }
gfCNCPoint5[17728] = {X 190.6670, Y 97.0659, Z -7.1667, A 0.000, B 0.000, C 0.000 }
gfCNCPoint5[17729] = {X 190.7727, Y 96.1162, Z -7.1667, A 0.000, B 0.000, C 0.000 }
gfCNCPoint5[17730] = {X 191.0846, Y 95.2129, Z -7.1667, A 0.000, B 0.000, C 0.000 }
gfCNCPoint5[17731] = {X 191.5874, Y 94.4003, Z -7.1667, A 0.000, B 0.000, C 0.000 }
gfCNCPoint5[17732] = {X 188.5647, Y 91.1002, Z -7.1667, A 0.000, B 0.000, C 0.000 }
gfCNCPoint5[17733] = {X 150.0898, Y 91.1002, Z -7.1667, A 0.000, B 0.000, C 0.000 }
gfCNCPoint5[17734] = {X 147.1456, Y 94.3621, Z -7.1667, A 0.000, B 0.000, C 0.000 }
gfCNCPoint5[17735] = {X 147.6648, Y 95.1835, Z -7.1667, A 0.000, B 0.000, C 0.000 }
gfCNCPoint5[17736] = {X 147.9881, Y 96.0999, Z -7.1667, A 0.000, B 0.000, C 0.000 }
gfCNCPoint5[17737] = {X 148.0991, Y 97.0653, Z -7.1667, A 0.000, B 0.000, C 0.000 }
gfCNCPoint5[17738] = {X 148.0991, Y 98.0000, Z -7.1667, A 0.000, B 0.000, C 0.000 }
gfCNCPoint5[17739] = {X 147.9908, Y 98.9613, Z -7.1667, A 0.000, B 0.000, C 0.000 }
gfCNCPoint5[17740] = {X 147.6713, Y 99.8744, Z -7.1667, A 0.000, B 0.000, C 0.000 }
gfCNCPoint5[17741] = {X 147.1566, Y 100.6935, Z -7.1667, A 0.000, B 0.000, C 0.000 }
gfCNCPoint5[17742] = {X 146.4726, Y 101.3775, Z -7.1667, A 0.000, B 0.000, C 0.000 }
gfCNCPoint5[17743] = {X 145.6535, Y 101.8922, Z -7.1667, A 0.000, B 0.000, C 0.000 }
gfCNCPoint5[17744] = {X 144.7404, Y 102.2117, Z -7.1667, A 0.000, B 0.000, C 0.000 }
gfCNCPoint5[17745] = {X 143.7791, Y 102.3200, Z -7.1667, A 0.000, B 0.000, C 0.000 }
gfCNCPoint5[17746] = {X 125.0000, Y 102.3200, Z -7.1667, A 0.000, B 0.000, C 0.000 }
gfCNCPoint5[17747] = {X 124.0387, Y 102.2117, Z -7.1667, A 0.000, B 0.000, C 0.000 }
gfCNCPoint5[17748] = {X 123.1256, Y 101.8922, Z -7.1667, A 0.000, B 0.000, C 0.000 }
gfCNCPoint5[17749] = {X 122.3065, Y 101.3775, Z -7.1667, A 0.000, B 0.000, C 0.000 }
gfCNCPoint5[17750] = {X 121.6225, Y 100.6935, Z -7.1667, A 0.000, B 0.000, C 0.000 }
gfCNCPoint5[17751] = {X 121.1078, Y 99.8744, Z -7.1667, A 0.000, B 0.000, C 0.000 }
gfCNCPoint5[17752] = {X 120.7883, Y 98.9613, Z -7.1667, A 0.000, B 0.000, C 0.000 }
gfCNCPoint5[17753] = {X 120.6800, Y 98.0000, Z -7.1667, A 0.000, B 0.000, C 0.000 }
gfCNCPoint5[17754] = {X 120.6800, Y 97.0659, Z -7.1667, A 0.000, B 0.000, C 0.000 }
gfCNCPoint5[17755] = {X 120.7831, Y 96.1277, Z -7.1667, A 0.000, B 0.000, C 0.000 }
gfCNCPoint5[17756] = {X 121.0876, Y 95.2342, Z -7.1667, A 0.000, B 0.000, C 0.000 }
gfCNCPoint5[17757] = {X 121.5788, Y 94.4281, Z -7.1667, A 0.000, B 0.000, C 0.000 }
gfCNCPoint5[17758] = {X 122.2334, Y 93.7480, Z -7.1667, A 0.000, B 0.000, C 0.000 }
gfCNCPoint5[17759] = {X 123.0201, Y 93.2264, Z -7.1667, A 0.000, B 0.000, C 0.000 }
gfCNCPoint5[17760] = {X 123.9013, Y 92.8880, Z -7.1667, A 0.000, B 0.000, C 0.000 }
gfCNCPoint5[17761] = {X 124.8350, Y 92.7491, Z -7.1667, A 0.000, B 0.000, C 0.000 }
gfCNCPoint5[17762] = {X 124.8802, Y 92.7312, Z -7.1667, A 0.000, B 0.000, C 0.000 }
gfCNCPoint5[17763] = {X 124.9277, Y 92.7205, Z -7.1667, A 0.000, B 0.000, C 0.000 }
gfCNCPoint5[17764] = {X 125.4500, Y 92.6430, Z -7.1667, A 0.000, B 0.000, C 0.000 }
gfCNCPoint5[17765] = {X 126.2807, Y 92.5032, Z -7.1667, A 0.000, B 0.000, C 0.000 }
gfCNCPoint5[17766] = {X 127.0999, Y 92.3069, Z -7.1667, A 0.000, B 0.000, C 0.000 }
gfCNCPoint5[17767] = {X 128.2870, Y 91.1908, Z -7.1667, A 0.000, B 0.000, C 0.000 }
gfCNCPoint5[17768] = {X 129.4114, Y 90.0115, Z -7.1667, A 0.000, B 0.000, C 0.000 }
gfCNCPoint5[17769] = {X 140.6794, Y 77.6384, Z -7.1667, A 0.000, B 0.000, C 0.000 }
gfCNCPoint5[17770] = {X 137.7220, Y 74.9452, Z -7.1667, A 0.000, B 0.000, C 0.000 }
gfCNCPoint5[17771] = {X 140.7385, Y 77.6923, Z -7.1667, A 0.000, B 0.000, C 0.000 }
gfCNCPoint5[17772] = {X 155.7322, Y 61.2282, Z -7.1667, A 0.000, B 0.000, C 0.000 }
gfCNCPoint5[17773] = {X 155.3666, Y 60.5221, Z -7.1667, A 0.000, B 0.000, C 0.000 }
gfCNCPoint5[17774] = {X 155.1392, Y 59.7601, Z -7.1667, A 0.000, B 0.000, C 0.000 }
gfCNCPoint5[17775] = {X 155.0581, Y 58.9691, Z -7.1667, A 0.000, B 0.000, C 0.000 }
gfCNCPoint5[17776] = {X 155.0580, Y 58.0000, Z -7.1667, A 0.000, B 0.000, C 0.000 }
gfCNCPoint5[17777] = {X 155.1643, Y 57.0565, Z -7.1667, A 0.000, B 0.000, C 0.000 }
gfCNCPoint5[17778] = {X 155.4778, Y 56.1603, Z -7.1667, A 0.000, B 0.000, C 0.000 }
gfCNCPoint5[17779] = {X 155.9830, Y 55.3564, Z -7.1667, A 0.000, B 0.000, C 0.000 }
gfCNCPoint5[17780] = {X 156.6544, Y 54.6850, Z -7.1667, A 0.000, B 0.000, C 0.000 }
gfCNCPoint5[17781] = {X 157.4583, Y 54.1799, Z -7.1667, A 0.000, B 0.000, C 0.000 }
gfCNCPoint5[17782] = {X 158.3545, Y 53.8663, Z -7.1667, A 0.000, B 0.000, C 0.000 }
gfCNCPoint5[17783] = {X 159.2980, Y 53.7600, Z -7.1667, A 0.000, B 0.000, C 0.000 }
gfCNCPoint5[17784] = {X 178.5335, Y 53.7600, Z -7.1667, A 0.000, B 0.000, C 0.000 }
gfCNCPoint5[17785] = {X 179.4770, Y 53.8663, Z -7.1667, A 0.000, B 0.000, C 0.000 }
gfCNCPoint5[17786] = {X 180.3732, Y 54.1799, Z -7.1667, A 0.000, B 0.000, C 0.000 }
gfCNCPoint5[17787] = {X 181.1771, Y 54.6850, Z -7.1667, A 0.000, B 0.000, C 0.000 }
gfCNCPoint5[17788] = {X 181.8485, Y 55.3564, Z -7.1667, A 0.000, B 0.000, C 0.000 }
gfCNCPoint5[17789] = {X 182.3536, Y 56.1603, Z -7.1667, A 0.000, B 0.000, C 0.000 }
gfCNCPoint5[17790] = {X 182.6672, Y 57.0565, Z -7.1667, A 0.000, B 0.000, C 0.000 }
gfCNCPoint5[17791] = {X 182.7735, Y 58.0000, Z -7.1667, A 0.000, B 0.000, C 0.000 }
gfCNCPoint5[17792] = {X 182.7735, Y 58.9342, Z -7.1667, A 0.000, B 0.000, C 0.000 }
gfCNCPoint5[17793] = {X 182.6985, Y 59.7281, Z -7.1667, A 0.000, B 0.000, C 0.000 }
gfCNCPoint5[17794] = {X 182.4761, Y 60.4940, Z -7.1667, A 0.000, B 0.000, C 0.000 }
gfCNCPoint5[17795] = {X 182.1143, Y 61.2046, Z -7.1667, A 0.000, B 0.000, C 0.000 }
gfCNCPoint5[17796] = {X 209.2374, Y 90.8137, Z -7.1667, A 0.000, B 0.000, C 0.000 }
gfCNCPoint5[17797] = {X 209.9114, Y 91.5117, Z -7.1667, A 0.000, B 0.000, C 0.000 }
gfCNCPoint5[17798] = {X 210.6211, Y 92.1735, Z -7.1667, A 0.000, B 0.000, C 0.000 }
gfCNCPoint5[17799] = {X 211.0313, Y 92.4511, Z -7.1667, A 0.000, B 0.000, C 0.000 }
gfCNCPoint5[17800] = {X 211.4989, Y 92.6147, Z -7.1667, A 0.000, B 0.000, C 0.000 }
gfCNCPoint5[17801] = {X 212.0943, Y 92.7400, Z -7.1667, A 0.000, B 0.000, C 0.000 }
gfCNCPoint5[17802] = {X 213.3841, Y 92.9001, Z -7.1667, A 0.000, B 0.000, C 0.000 }
gfCNCPoint5[17803] = {X 214.4459, Y 92.8161, Z -7.1667, A 0.000, B 0.000, C 0.000 }
gfCNCPoint5[17804] = {X 215.5093, Y 92.7545, Z -7.1667, A 0.000, B 0.000, C 0.000 }
gfCNCPoint5[17805] = {X 216.1939, Y 92.6799, Z -7.1667, A 0.000, B 0.000, C 0.000 }
gfCNCPoint5[17806] = {X 216.8530, Y 92.4805, Z -7.1667, A 0.000, B 0.000, C 0.000 }
gfCNCPoint5[17807] = {X 217.4643, Y 92.1634, Z -7.1667, A 0.000, B 0.000, C 0.000 }
gfCNCPoint5[17808] = {X 223.0046, Y 88.5879, Z -7.1667, A 0.000, B 0.000, C 0.000 }
gfCNCPoint5[17809] = {X 246.0024, Y 73.8825, Z -7.1667, A 0.000, B 0.000, C 0.000 }
gfCNCPoint5[17810] = {X 221.6603, Y 64.3304, Z -7.1667, A 0.000, B 0.000, C 0.000 }
gfCNCPoint5[17811] = {X 219.8841, Y 63.7361, Z -7.1667, A 0.000, B 0.000, C 0.000 }
gfCNCPoint5[17812] = {X 218.0517, Y 63.3481, Z -7.1667, A 0.000, B 0.000, C 0.000 }
gfCNCPoint5[17813] = {X 216.1870, Y 63.1716, Z -7.1667, A 0.000, B 0.000, C 0.000 }
gfCNCPoint5[17814] = {X 215.2724, Y 63.0398, Z -7.1667, A 0.000, B 0.000, C 0.000 }
gfCNCPoint5[17815] = {X 214.4080, Y 62.7130, Z -7.1667, A 0.000, B 0.000, C 0.000 }
gfCNCPoint5[17816] = {X 213.6350, Y 62.2067, Z -7.1667, A 0.000, B 0.000, C 0.000 }
gfCNCPoint5[17817] = {X 212.9900, Y 61.5450, Z -7.1667, A 0.000, B 0.000, C 0.000 }
gfCNCPoint5[17818] = {X 212.5037, Y 60.7592, Z -7.1667, A 0.000, B 0.000, C 0.000 }
gfCNCPoint5[17819] = {X 212.1992, Y 59.8868, Z -7.1667, A 0.000, B 0.000, C 0.000 }
gfCNCPoint5[17820] = {X 212.0910, Y 58.9691, Z -7.1667, A 0.000, B 0.000, C 0.000 }
gfCNCPoint5[17821] = {X 212.0908, Y 58.0000, Z -7.1667, A 0.000, B 0.000, C 0.000 }
gfCNCPoint5[17822] = {X 212.1971, Y 57.0565, Z -7.1667, A 0.000, B 0.000, C 0.000 }
gfCNCPoint5[17823] = {X 212.5107, Y 56.1603, Z -7.1667, A 0.000, B 0.000, C 0.000 }
gfCNCPoint5[17824] = {X 213.0158, Y 55.3564, Z -7.1667, A 0.000, B 0.000, C 0.000 }
gfCNCPoint5[17825] = {X 213.6872, Y 54.6850, Z -7.1667, A 0.000, B 0.000, C 0.000 }
gfCNCPoint5[17826] = {X 214.4911, Y 54.1799, Z -7.1667, A 0.000, B 0.000, C 0.000 }
gfCNCPoint5[17827] = {X 215.3873, Y 53.8663, Z -7.1667, A 0.000, B 0.000, C 0.000 }
gfCNCPoint5[17828] = {X 216.3308, Y 53.7600, Z -7.1667, A 0.000, B 0.000, C 0.000 }
gfCNCPoint5[17829] = {X 237.2617, Y 53.7600, Z -7.1667, A 0.000, B 0.000, C 0.000 }
gfCNCPoint5[17830] = {X 238.2052, Y 53.8663, Z -7.1667, A 0.000, B 0.000, C 0.000 }
gfCNCPoint5[17831] = {X 239.1014, Y 54.1799, Z -7.1667, A 0.000, B 0.000, C 0.000 }
gfCNCPoint5[17832] = {X 239.9053, Y 54.6850, Z -7.1667, A 0.000, B 0.000, C 0.000 }
gfCNCPoint5[17833] = {X 240.5767, Y 55.3564, Z -7.1667, A 0.000, B 0.000, C 0.000 }
gfCNCPoint5[17834] = {X 241.0818, Y 56.1603, Z -7.1667, A 0.000, B 0.000, C 0.000 }
gfCNCPoint5[17835] = {X 241.3954, Y 57.0565, Z -7.1667, A 0.000, B 0.000, C 0.000 }
gfCNCPoint5[17836] = {X 241.5017, Y 58.0000, Z -7.1667, A 0.000, B 0.000, C 0.000 }
gfCNCPoint5[17837] = {X 241.5017, Y 58.2864, Z -7.1667, A 0.000, B 0.000, C 0.000 }
gfCNCPoint5[17838] = {X 248.0855, Y 60.8537, Z -7.1667, A 0.000, B 0.000, C 0.000 }
gfCNCPoint5[17839] = {X 275.7119, Y 71.8192, Z -7.1667, A 0.000, B 0.000, C 0.000 }
gfCNCPoint5[17840] = {X 275.7135, Y 63.1422, Z -7.1667, A 0.000, B 0.000, C 0.000 }
gfCNCPoint5[17841] = {X 274.8650, Y 62.9474, Z -7.1667, A 0.000, B 0.000, C 0.000 }
gfCNCPoint5[17842] = {X 274.0741, Y 62.5835, Z -7.1667, A 0.000, B 0.000, C 0.000 }
gfCNCPoint5[17843] = {X 273.3743, Y 62.0657, Z -7.1667, A 0.000, B 0.000, C 0.000 }
gfCNCPoint5[17844] = {X 272.7950, Y 61.4159, Z -7.1667, A 0.000, B 0.000, C 0.000 }
gfCNCPoint5[17845] = {X 272.3605, Y 60.6615, Z -7.1667, A 0.000, B 0.000, C 0.000 }
gfCNCPoint5[17846] = {X 272.0894, Y 59.8343, Z -7.1667, A 0.000, B 0.000, C 0.000 }
gfCNCPoint5[17847] = {X 271.9928, Y 58.9691, Z -7.1667, A 0.000, B 0.000, C 0.000 }
gfCNCPoint5[17848] = {X 271.9927, Y 58.0000, Z -7.1667, A 0.000, B 0.000, C 0.000 }
gfCNCPoint5[17849] = {X 272.0990, Y 57.0565, Z -7.1667, A 0.000, B 0.000, C 0.000 }
gfCNCPoint5[17850] = {X 272.4126, Y 56.1603, Z -7.1667, A 0.000, B 0.000, C 0.000 }
gfCNCPoint5[17851] = {X 272.9177, Y 55.3564, Z -7.1667, A 0.000, B 0.000, C 0.000 }
gfCNCPoint5[17852] = {X 273.5891, Y 54.6850, Z -7.1667, A 0.000, B 0.000, C 0.000 }
gfCNCPoint5[17853] = {X 274.3930, Y 54.1799, Z -7.1667, A 0.000, B 0.000, C 0.000 }
gfCNCPoint5[17854] = {X 275.2892, Y 53.8663, Z -7.1667, A 0.000, B 0.000, C 0.000 }
gfCNCPoint5[17855] = {X 276.2327, Y 53.7600, Z -7.1667, A 0.000, B 0.000, C 0.000 }
gfCNCPoint5[17856] = {X 292.7731, Y 53.7600, Z -7.1667, A 0.000, B 0.000, C 0.000 }
gfCNCPoint5[17857] = {X 293.7166, Y 53.8663, Z -7.1667, A 0.000, B 0.000, C 0.000 }
gfCNCPoint5[17858] = {X 294.6128, Y 54.1799, Z -7.1667, A 0.000, B 0.000, C 0.000 }
gfCNCPoint5[17859] = {X 295.4167, Y 54.6850, Z -7.1667, A 0.000, B 0.000, C 0.000 }
gfCNCPoint5[17860] = {X 296.0881, Y 55.3564, Z -7.1667, A 0.000, B 0.000, C 0.000 }
gfCNCPoint5[17861] = {X 296.5932, Y 56.1603, Z -7.1667, A 0.000, B 0.000, C 0.000 }
gfCNCPoint5[17862] = {X 296.9068, Y 57.0565, Z -7.1667, A 0.000, B 0.000, C 0.000 }
gfCNCPoint5[17863] = {X 297.0131, Y 58.0000, Z -7.1667, A 0.000, B 0.000, C 0.000 }
gfCNCPoint5[17864] = {X 297.0131, Y 58.9348, Z -7.1667, A 0.000, B 0.000, C 0.000 }
gfCNCPoint5[17865] = {X 296.9208, Y 59.8046, Z -7.1667, A 0.000, B 0.000, C 0.000 }
gfCNCPoint5[17866] = {X 296.6527, Y 60.6371, Z -7.1667, A 0.000, B 0.000, C 0.000 }
gfCNCPoint5[17867] = {X 296.2200, Y 61.3973, Z -7.1667, A 0.000, B 0.000, C 0.000 }
gfCNCPoint5[17868] = {X 295.6411, Y 62.0529, Z -7.1667, A 0.000, B 0.000, C 0.000 }
gfCNCPoint5[17869] = {X 294.9403, Y 62.5764, Z -7.1667, A 0.000, B 0.000, C 0.000 }
gfCNCPoint5[17870] = {X 294.1474, Y 62.9456, Z -7.1667, A 0.000, B 0.000, C 0.000 }
gfCNCPoint5[17871] = {X 293.2957, Y 63.1448, Z -7.1667, A 0.000, B 0.000, C 0.000 }
gfCNCPoint5[17872] = {X 293.3049, Y 92.8496, Z -7.1667, A 0.000, B 0.000, C 0.000 }
gfCNCPoint5[17873] = {X 294.1545, Y 93.0529, Z -7.1667, A 0.000, B 0.000, C 0.000 }
gfCNCPoint5[17874] = {X 294.9449, Y 93.4247, Z -7.1667, A 0.000, B 0.000, C 0.000 }
gfCNCPoint5[17875] = {X 295.6432, Y 93.9495, Z -7.1667, A 0.000, B 0.000, C 0.000 }
gfCNCPoint5[17876] = {X 296.2202, Y 94.6054, Z -7.1667, A 0.000, B 0.000, C 0.000 }
gfCNCPoint5[17877] = {X 296.6517, Y 95.3649, Z -7.1667, A 0.000, B 0.000, C 0.000 }
gfCNCPoint5[17878] = {X 296.9198, Y 96.1964, Z -7.1667, A 0.000, B 0.000, C 0.000 }
gfCNCPoint5[17879] = {X 297.0131, Y 97.0649, Z -7.1667, A 0.000, B 0.000, C 0.000 }
gfCNCPoint5[17880] = {X 297.0131, Y 98.0000, Z -7.1667, A 0.000, B 0.000, C 0.000 }
gfCNCPoint5[17881] = {X 296.9068, Y 98.9435, Z -7.1667, A 0.000, B 0.000, C 0.000 }
gfCNCPoint5[17882] = {X 296.5932, Y 99.8397, Z -7.1667, A 0.000, B 0.000, C 0.000 }
gfCNCPoint5[17883] = {X 296.0881, Y 100.6436, Z -7.1667, A 0.000, B 0.000, C 0.000 }
gfCNCPoint5[17884] = {X 295.4167, Y 101.3150, Z -7.1667, A 0.000, B 0.000, C 0.000 }
gfCNCPoint5[17885] = {X 294.6128, Y 101.8201, Z -7.1667, A 0.000, B 0.000, C 0.000 }
gfCNCPoint5[17886] = {X 293.7166, Y 102.1337, Z -7.1667, A 0.000, B 0.000, C 0.000 }
gfCNCPoint5[17887] = {X 292.7731, Y 102.2400, Z -7.1667, A 0.000, B 0.000, C 0.000 }
gfCNCPoint5[17888] = {X 276.2327, Y 102.2400, Z -7.1667, A 0.000, B 0.000, C 0.000 }
gfCNCPoint5[17889] = {X 275.2892, Y 102.1337, Z -7.1667, A 0.000, B 0.000, C 0.000 }
gfCNCPoint5[17890] = {X 274.3930, Y 101.8201, Z -7.1667, A 0.000, B 0.000, C 0.000 }
gfCNCPoint5[17891] = {X 273.5891, Y 101.3150, Z -7.1667, A 0.000, B 0.000, C 0.000 }
gfCNCPoint5[17892] = {X 272.9177, Y 100.6436, Z -7.1667, A 0.000, B 0.000, C 0.000 }
gfCNCPoint5[17893] = {X 272.4126, Y 99.8397, Z -7.1667, A 0.000, B 0.000, C 0.000 }
gfCNCPoint5[17894] = {X 272.0990, Y 98.9435, Z -7.1667, A 0.000, B 0.000, C 0.000 }
gfCNCPoint5[17895] = {X 271.9927, Y 98.0000, Z -7.1667, A 0.000, B 0.000, C 0.000 }
gfCNCPoint5[17896] = {X 271.9927, Y 97.0658, Z -7.1667, A 0.000, B 0.000, C 0.000 }
gfCNCPoint5[17897] = {X 272.0830, Y 96.1956, Z -7.1667, A 0.000, B 0.000, C 0.000 }
gfCNCPoint5[17898] = {X 272.3500, Y 95.3624, Z -7.1667, A 0.000, B 0.000, C 0.000 }
gfCNCPoint5[17899] = {X 272.7823, Y 94.6017, Z -7.1667, A 0.000, B 0.000, C 0.000 }
gfCNCPoint5[17900] = {X 273.3615, Y 93.9460, Z -7.1667, A 0.000, B 0.000, C 0.000 }
gfCNCPoint5[17901] = {X 274.0630, Y 93.4231, Z -7.1667, A 0.000, B 0.000, C 0.000 }
gfCNCPoint5[17902] = {X 274.8569, Y 93.0553, Z -7.1667, A 0.000, B 0.000, C 0.000 }
gfCNCPoint5[17903] = {X 275.7094, Y 92.8584, Z -7.1667, A 0.000, B 0.000, C 0.000 }
gfCNCPoint5[17904] = {X 275.7094, Y 85.5404, Z -7.1667, A 0.000, B 0.000, C 0.000 }
gfCNCPoint5[17905] = {X 262.6314, Y 80.4138, Z -7.1667, A 0.000, B 0.000, C 0.000 }
gfCNCPoint5[17906] = {X 262.2351, Y 80.6641, Z -7.1667, A 0.000, B 0.000, C 0.000 }
gfCNCPoint5[17907] = {X 237.7172, Y 96.5450, Z -7.1667, A 0.000, B 0.000, C 0.000 }
gfCNCPoint5[17908] = {X 237.7198, Y 97.0653, Z -7.1667, A 0.000, B 0.000, C 0.000 }
gfCNCPoint5[17909] = {X 237.7198, Y 98.0000, Z -7.1667, A 0.000, B 0.000, C 0.000 }
gfCNCPoint5[17910] = {X 237.6135, Y 98.9435, Z -7.1667, A 0.000, B 0.000, C 0.000 }
gfCNCPoint5[17911] = {X 237.2999, Y 99.8397, Z -7.1667, A 0.000, B 0.000, C 0.000 }
gfCNCPoint5[17912] = {X 236.7948, Y 100.6436, Z -7.1667, A 0.000, B 0.000, C 0.000 }
gfCNCPoint5[17913] = {X 236.1234, Y 101.3150, Z -7.1667, A 0.000, B 0.000, C 0.000 }
gfCNCPoint5[17914] = {X 235.3195, Y 101.8201, Z -7.1667, A 0.000, B 0.000, C 0.000 }
gfCNCPoint5[17915] = {X 234.4233, Y 102.1337, Z -7.1667, A 0.000, B 0.000, C 0.000 }
gfCNCPoint5[17916] = {X 233.4798, Y 102.2400, Z -7.1667, A 0.000, B 0.000, C 0.000 }
gfCNCPoint5[17917] = {X 214.1790, Y 102.2400, Z -7.1667, A 0.000, B 0.000, C 0.000 }
gfCNCPoint5[17918] = {X 213.7861, Y 102.2218, Z -7.1667, A 0.000, B 0.000, C 0.000 }
gfCNCPoint5[17919] = {X 213.3966, Y 102.1672, Z -7.1667, A 0.000, B 0.000, C 0.000 }
gfCNCPoint5[17920] = {X 213.0070, Y 102.2218, Z -7.1667, A 0.000, B 0.000, C 0.000 }
gfCNCPoint5[17921] = {X 212.6141, Y 102.2400, Z -7.1667, A 0.000, B 0.000, C 0.000 }
gfCNCPoint5[17922] = {X 194.9870, Y 102.2400, Z -7.1667, A 0.000, B 0.000, C 0.000 }
gfCNCPoint5[17923] = {X 194.0435, Y 102.1337, Z -7.1667, A 0.000, B 0.000, C 0.000 }
gfCNCPoint5[17924] = {X 193.1473, Y 101.8201, Z -7.1667, A 0.000, B 0.000, C 0.000 }
gfCNCPoint5[17925] = {X 192.3434, Y 101.3150, Z -7.1667, A 0.000, B 0.000, C 0.000 }
gfCNCPoint5[17926] = {X 191.6720, Y 100.6436, Z -7.1667, A 0.000, B 0.000, C 0.000 }
gfCNCPoint5[17927] = {X 191.1669, Y 99.8397, Z -7.1667, A 0.000, B 0.000, C 0.000 }
gfCNCPoint5[17928] = {X 190.8533, Y 98.9435, Z -7.1667, A 0.000, B 0.000, C 0.000 }
gfCNCPoint5[17929] = {X 190.7470, Y 98.0000, Z -7.1667, A 0.000, B 0.000, C 0.000 }
gfCNCPoint5[17930] = {X 190.7470, Y 97.0659, Z -7.1667, A 0.000, B 0.000, C 0.000 }
gfCNCPoint5[17931] = {X 190.8557, Y 96.1118, Z -7.1667, A 0.000, B 0.000, C 0.000 }
gfCNCPoint5[17932] = {X 191.1764, Y 95.2065, Z -7.1667, A 0.000, B 0.000, C 0.000 }
gfCNCPoint5[17933] = {X 191.6926, Y 94.3967, Z -7.1667, A 0.000, B 0.000, C 0.000 }
gfCNCPoint5[17934] = {X 188.5999, Y 91.0202, Z -7.1667, A 0.000, B 0.000, C 0.000 }
gfCNCPoint5[17935] = {X 150.0543, Y 91.0202, Z -7.1667, A 0.000, B 0.000, C 0.000 }
gfCNCPoint5[17936] = {X 147.0402, Y 94.3594, Z -7.1667, A 0.000, B 0.000, C 0.000 }
gfCNCPoint5[17937] = {X 147.5729, Y 95.1777, Z -7.1667, A 0.000, B 0.000, C 0.000 }
gfCNCPoint5[17938] = {X 147.9050, Y 96.0958, Z -7.1667, A 0.000, B 0.000, C 0.000 }
gfCNCPoint5[17939] = {X 148.0191, Y 97.0655, Z -7.1667, A 0.000, B 0.000, C 0.000 }
gfCNCPoint5[17940] = {X 148.0191, Y 98.0000, Z -7.1667, A 0.000, B 0.000, C 0.000 }
gfCNCPoint5[17941] = {X 147.9128, Y 98.9435, Z -7.1667, A 0.000, B 0.000, C 0.000 }
gfCNCPoint5[17942] = {X 147.5992, Y 99.8397, Z -7.1667, A 0.000, B 0.000, C 0.000 }
gfCNCPoint5[17943] = {X 147.0941, Y 100.6436, Z -7.1667, A 0.000, B 0.000, C 0.000 }
gfCNCPoint5[17944] = {X 146.4227, Y 101.3150, Z -7.1667, A 0.000, B 0.000, C 0.000 }
gfCNCPoint5[17945] = {X 145.6188, Y 101.8201, Z -7.1667, A 0.000, B 0.000, C 0.000 }
gfCNCPoint5[17946] = {X 144.7226, Y 102.1337, Z -7.1667, A 0.000, B 0.000, C 0.000 }
gfCNCPoint5[17947] = {X 143.7791, Y 102.2400, Z -7.1667, A 0.000, B 0.000, C 0.000 }
gfCNCPoint5[17948] = {X 125.0000, Y 102.2400, Z -7.1667, A 0.000, B 0.000, C 0.000 }
gfCNCPoint5[17949] = {X 124.0565, Y 102.1337, Z -7.1667, A 0.000, B 0.000, C 0.000 }
gfCNCPoint5[17950] = {X 123.1603, Y 101.8201, Z -7.1667, A 0.000, B 0.000, C 0.000 }
gfCNCPoint5[17951] = {X 122.3564, Y 101.3150, Z -7.1667, A 0.000, B 0.000, C 0.000 }
gfCNCPoint5[17952] = {X 121.6850, Y 100.6436, Z -7.1667, A 0.000, B 0.000, C 0.000 }
gfCNCPoint5[17953] = {X 121.1799, Y 99.8397, Z -7.1667, A 0.000, B 0.000, C 0.000 }
gfCNCPoint5[17954] = {X 120.8663, Y 98.9435, Z -7.1667, A 0.000, B 0.000, C 0.000 }
gfCNCPoint5[17955] = {X 120.7600, Y 98.0000, Z -7.1667, A 0.000, B 0.000, C 0.000 }
gfCNCPoint5[17956] = {X 120.7600, Y 97.0659, Z -7.1667, A 0.000, B 0.000, C 0.000 }
gfCNCPoint5[17957] = {X 120.8618, Y 96.1425, Z -7.1667, A 0.000, B 0.000, C 0.000 }
gfCNCPoint5[17958] = {X 121.1622, Y 95.2634, Z -7.1667, A 0.000, B 0.000, C 0.000 }
gfCNCPoint5[17959] = {X 121.6469, Y 94.4709, Z -7.1667, A 0.000, B 0.000, C 0.000 }
gfCNCPoint5[17960] = {X 122.2925, Y 93.8029, Z -7.1667, A 0.000, B 0.000, C 0.000 }
gfCNCPoint5[17961] = {X 123.0682, Y 93.2916, Z -7.1667, A 0.000, B 0.000, C 0.000 }
gfCNCPoint5[17962] = {X 123.9365, Y 92.9615, Z -7.1667, A 0.000, B 0.000, C 0.000 }
gfCNCPoint5[17963] = {X 124.8560, Y 92.8284, Z -7.1667, A 0.000, B 0.000, C 0.000 }
gfCNCPoint5[17964] = {X 124.8964, Y 92.8101, Z -7.1667, A 0.000, B 0.000, C 0.000 }
gfCNCPoint5[17965] = {X 124.9395, Y 92.7996, Z -7.1667, A 0.000, B 0.000, C 0.000 }
gfCNCPoint5[17966] = {X 125.4612, Y 92.7222, Z -7.1667, A 0.000, B 0.000, C 0.000 }
gfCNCPoint5[17967] = {X 126.3061, Y 92.5797, Z -7.1667, A 0.000, B 0.000, C 0.000 }
gfCNCPoint5[17968] = {X 127.1392, Y 92.3790, Z -7.1667, A 0.000, B 0.000, C 0.000 }
gfCNCPoint5[17969] = {X 128.3368, Y 91.2541, Z -7.1667, A 0.000, B 0.000, C 0.000 }
gfCNCPoint5[17970] = {X 129.4708, Y 90.0651, Z -7.1667, A 0.000, B 0.000, C 0.000 }
gfCNCPoint5[17971] = {X 140.7385, Y 77.6923, Z -7.1667, A 0.000, B 0.000, C 0.000 }
gfCNCPoint5[17972] = {X 137.7811, Y 74.9990, Z -7.1667, A 0.000, B 0.000, C 0.000 }
gfCNCPoint5[17973] = {X 140.7977, Y 77.7462, Z -7.1667, A 0.000, B 0.000, C 0.000 }
gfCNCPoint5[17974] = {X 155.8331, Y 61.2363, Z -7.1667, A 0.000, B 0.000, C 0.000 }
gfCNCPoint5[17975] = {X 155.4563, Y 60.5300, Z -7.1667, A 0.000, B 0.000, C 0.000 }
gfCNCPoint5[17976] = {X 155.2217, Y 59.7646, Z -7.1667, A 0.000, B 0.000, C 0.000 }
gfCNCPoint5[17977] = {X 155.1381, Y 58.9684, Z -7.1667, A 0.000, B 0.000, C 0.000 }
gfCNCPoint5[17978] = {X 155.1380, Y 58.0000, Z -7.1667, A 0.000, B 0.000, C 0.000 }
gfCNCPoint5[17979] = {X 155.2423, Y 57.0743, Z -7.1667, A 0.000, B 0.000, C 0.000 }
gfCNCPoint5[17980] = {X 155.5499, Y 56.1950, Z -7.1667, A 0.000, B 0.000, C 0.000 }
gfCNCPoint5[17981] = {X 156.0455, Y 55.4063, Z -7.1667, A 0.000, B 0.000, C 0.000 }
gfCNCPoint5[17982] = {X 156.7042, Y 54.7476, Z -7.1667, A 0.000, B 0.000, C 0.000 }
gfCNCPoint5[17983] = {X 157.4930, Y 54.2520, Z -7.1667, A 0.000, B 0.000, C 0.000 }
gfCNCPoint5[17984] = {X 158.3723, Y 53.9443, Z -7.1667, A 0.000, B 0.000, C 0.000 }
gfCNCPoint5[17985] = {X 159.2980, Y 53.8400, Z -7.1667, A 0.000, B 0.000, C 0.000 }
gfCNCPoint5[17986] = {X 178.5335, Y 53.8400, Z -7.1667, A 0.000, B 0.000, C 0.000 }
gfCNCPoint5[17987] = {X 179.4592, Y 53.9443, Z -7.1667, A 0.000, B 0.000, C 0.000 }
gfCNCPoint5[17988] = {X 180.3385, Y 54.2520, Z -7.1667, A 0.000, B 0.000, C 0.000 }
gfCNCPoint5[17989] = {X 181.1272, Y 54.7476, Z -7.1667, A 0.000, B 0.000, C 0.000 }
gfCNCPoint5[17990] = {X 181.7859, Y 55.4063, Z -7.1667, A 0.000, B 0.000, C 0.000 }
gfCNCPoint5[17991] = {X 182.2815, Y 56.1950, Z -7.1667, A 0.000, B 0.000, C 0.000 }
gfCNCPoint5[17992] = {X 182.5892, Y 57.0743, Z -7.1667, A 0.000, B 0.000, C 0.000 }
gfCNCPoint5[17993] = {X 182.6935, Y 58.0000, Z -7.1667, A 0.000, B 0.000, C 0.000 }
gfCNCPoint5[17994] = {X 182.6935, Y 58.9342, Z -7.1667, A 0.000, B 0.000, C 0.000 }
gfCNCPoint5[17995] = {X 182.6160, Y 59.7332, Z -7.1667, A 0.000, B 0.000, C 0.000 }
gfCNCPoint5[17996] = {X 182.3866, Y 60.5024, Z -7.1667, A 0.000, B 0.000, C 0.000 }
gfCNCPoint5[17997] = {X 182.0136, Y 61.2132, Z -7.1667, A 0.000, B 0.000, C 0.000 }
gfCNCPoint5[17998] = {X 209.1784, Y 90.8677, Z -7.1667, A 0.000, B 0.000, C 0.000 }
gfCNCPoint5[17999] = {X 209.8553, Y 91.5688, Z -7.1667, A 0.000, B 0.000, C 0.000 }
gfCNCPoint5[18000] = {X 210.5681, Y 92.2334, Z -7.1667, A 0.000, B 0.000, C 0.000 }
gfCNCPoint5[18001] = {X 210.9954, Y 92.5226, Z -7.1667, A 0.000, B 0.000, C 0.000 }
gfCNCPoint5[18002] = {X 211.4824, Y 92.6930, Z -7.1667, A 0.000, B 0.000, C 0.000 }
gfCNCPoint5[18003] = {X 212.0811, Y 92.8190, Z -7.1667, A 0.000, B 0.000, C 0.000 }
gfCNCPoint5[18004] = {X 213.3842, Y 92.9831, Z -7.1667, A 0.000, B 0.000, C 0.000 }
gfCNCPoint5[18005] = {X 213.3985, Y 92.9791, Z -7.1667, A 0.000, B 0.000, C 0.000 }
gfCNCPoint5[18006] = {X 214.4544, Y 92.8957, Z -7.1667, A 0.000, B 0.000, C 0.000 }
gfCNCPoint5[18007] = {X 215.5118, Y 92.8345, Z -7.1667, A 0.000, B 0.000, C 0.000 }
gfCNCPoint5[18008] = {X 216.2107, Y 92.7581, Z -7.1667, A 0.000, B 0.000, C 0.000 }
gfCNCPoint5[18009] = {X 216.8836, Y 92.5544, Z -7.1667, A 0.000, B 0.000, C 0.000 }
gfCNCPoint5[18010] = {X 217.5076, Y 92.2306, Z -7.1667, A 0.000, B 0.000, C 0.000 }
gfCNCPoint5[18011] = {X 223.0478, Y 88.6552, Z -7.1667, A 0.000, B 0.000, C 0.000 }
gfCNCPoint5[18012] = {X 246.1777, Y 73.8654, Z -7.1667, A 0.000, B 0.000, C 0.000 }
gfCNCPoint5[18013] = {X 221.6900, Y 64.2562, Z -7.1667, A 0.000, B 0.000, C 0.000 }
gfCNCPoint5[18014] = {X 219.9051, Y 63.6589, Z -7.1667, A 0.000, B 0.000, C 0.000 }
gfCNCPoint5[18015] = {X 218.0637, Y 63.2690, Z -7.1667, A 0.000, B 0.000, C 0.000 }
gfCNCPoint5[18016] = {X 216.1900, Y 63.0917, Z -7.1667, A 0.000, B 0.000, C 0.000 }
gfCNCPoint5[18017] = {X 215.2926, Y 62.9624, Z -7.1667, A 0.000, B 0.000, C 0.000 }
gfCNCPoint5[18018] = {X 214.4445, Y 62.6418, Z -7.1667, A 0.000, B 0.000, C 0.000 }
gfCNCPoint5[18019] = {X 213.6860, Y 62.1451, Z -7.1667, A 0.000, B 0.000, C 0.000 }
gfCNCPoint5[18020] = {X 213.0531, Y 61.4958, Z -7.1667, A 0.000, B 0.000, C 0.000 }
gfCNCPoint5[18021] = {X 212.5760, Y 60.7249, Z -7.1667, A 0.000, B 0.000, C 0.000 }
gfCNCPoint5[18022] = {X 212.2772, Y 59.8688, Z -7.1667, A 0.000, B 0.000, C 0.000 }
gfCNCPoint5[18023] = {X 212.1710, Y 58.9684, Z -7.1667, A 0.000, B 0.000, C 0.000 }
gfCNCPoint5[18024] = {X 212.1708, Y 58.0000, Z -7.1667, A 0.000, B 0.000, C 0.000 }
gfCNCPoint5[18025] = {X 212.2751, Y 57.0743, Z -7.1667, A 0.000, B 0.000, C 0.000 }
gfCNCPoint5[18026] = {X 212.5828, Y 56.1950, Z -7.1667, A 0.000, B 0.000, C 0.000 }
gfCNCPoint5[18027] = {X 213.0784, Y 55.4063, Z -7.1667, A 0.000, B 0.000, C 0.000 }
gfCNCPoint5[18028] = {X 213.7371, Y 54.7476, Z -7.1667, A 0.000, B 0.000, C 0.000 }
gfCNCPoint5[18029] = {X 214.5259, Y 54.2520, Z -7.1667, A 0.000, B 0.000, C 0.000 }
gfCNCPoint5[18030] = {X 215.4051, Y 53.9443, Z -7.1667, A 0.000, B 0.000, C 0.000 }
gfCNCPoint5[18031] = {X 216.3308, Y 53.8400, Z -7.1667, A 0.000, B 0.000, C 0.000 }
gfCNCPoint5[18032] = {X 237.2617, Y 53.8400, Z -7.1667, A 0.000, B 0.000, C 0.000 }
gfCNCPoint5[18033] = {X 238.1874, Y 53.9443, Z -7.1667, A 0.000, B 0.000, C 0.000 }
gfCNCPoint5[18034] = {X 239.0666, Y 54.2520, Z -7.1667, A 0.000, B 0.000, C 0.000 }
gfCNCPoint5[18035] = {X 239.8554, Y 54.7476, Z -7.1667, A 0.000, B 0.000, C 0.000 }
gfCNCPoint5[18036] = {X 240.5141, Y 55.4063, Z -7.1667, A 0.000, B 0.000, C 0.000 }
gfCNCPoint5[18037] = {X 241.0097, Y 56.1950, Z -7.1667, A 0.000, B 0.000, C 0.000 }
gfCNCPoint5[18038] = {X 241.3174, Y 57.0743, Z -7.1667, A 0.000, B 0.000, C 0.000 }
gfCNCPoint5[18039] = {X 241.4217, Y 58.0000, Z -7.1667, A 0.000, B 0.000, C 0.000 }
gfCNCPoint5[18040] = {X 241.4217, Y 58.3411, Z -7.1667, A 0.000, B 0.000, C 0.000 }
